// TwinCAT 3 PLC project HAWino
// ProgramVersion: 3.1.4026.19
// libraries:
//   Tc2_Math, * (Beckhoff Automation GmbH)
//   Tc2_Standard, * (Beckhoff Automation GmbH)
//   Tc2_System, * (Beckhoff Automation GmbH)
//   Tc2_Utilities, * (Beckhoff Automation GmbH)
//   Tc3_IotBase, * (Beckhoff Automation GmbH)
//   Tc3_JsonXml, * (Beckhoff Automation GmbH)
//   Tc3_Module, * (Beckhoff Automation GmbH)
// project tree:
//   / BahnplanungTask.TcTTO, MotorTask.TcTTO, PlcTask.TcTTO, SOCTask.TcTTO
//   DUTs/Gewerk 2/ E_RobotState.TcDUT, sCmd.TcDUT, sError.TcDUT, sFahrvektor.TcDUT, sGeneralState.TcDUT, sJob.TcDUT, sJobState.TcDUT, sKoordinate.TcDUT, sMqttIn.TcDUT, sMqttOut.TcDUT, sPosition.TcDUT, sStatesForTest.TcDUT, sToken.TcDUT
//   DUTs/Gewerk 3/ Bumperstatus.TcDUT, EKF_Data.TcDUT, GripperCmd_Enum.TcDUT, Position.TcDUT, ReglerState.TcDUT, RobotControl.TcDUT, RobotStatus.TcDUT, WheelVelocity.TcDUT
//   DUTs/PowerManagement/ FleetManagement.TcDUT, ST_PwrMgmt_HAWino.TcDUT, ST_PwrMgmt_HAWino_In.TcDUT, ST_PwrMgmt_HAWino_Out.TcDUT
//   DUTs/Sys/ CoreDriveState.TcDUT, CoreGripperControlState.TcDUT, DUT_SysState.TcDUT, RobotInternalData.TcDUT, RobotPose.TcDUT, U_IpAdr.TcDUT
//   GVLs/ CollisionDetection.TcGVL, GVL_Gripper.TcGVL, GVL_Maps.TcGVL, GVL_RobotConstant.TcGVL, GVL_Datatransfer23.TcGVL, GVL_RobotCoordinates.TcGVL, MQTT_Bahnplanung_Sync.TcGVL, Var_HAWIno.TcGVL
//   POUs/HAWinoCore/001_MotorTask/ FB_Drehzahlregler.TcPOU, Main_MotorTask.TcPOU, FB_Positionsregler.TcPOU
//   POUs/HAWinoCore/01_Motors/ Bumper.TcPOU, Gripper.TcPOU
//   POUs/HAWinoCore/03_Communication/ Camera.TcPOU, CameraConnectionUDP.TcPOU, MQTT.TcPOU
//   POUs/HAWinoCore/02_IR-Sensors/ IrDistanceFromRaw.TcPOU, IrDistanceSensors.TcPOU
//   POUs/HAWinoCore/04_SystemManagment/ FKT_Scale.TcPOU, PowerManager.TcPOU
//   POUs/HAWinoCore/05_Bahnplanung/ FB_AngleMap.TcPOU, FB_CollisionAvoidance.TcPOU, FB_CollisionAvoidanceV2.TcPOU, FB_CollisionAvoidanceV22.TcPOU, FB_CollisionAvoidanceV3.TcPOU, FB_CollisionAvoidanceV3_4.TcPOU, FB_Mapping.TcPOU, FB_MQTT.TcPOU, FB_MQTTNeu.TcPOU, FB_Navigation.TcPOU, FB_RobotStateMachine.TcPOU, FB_StatesTest.TcPOU, FC_ATAN2.TcPOU, Main_Bahnplanung.TcPOU
//   POUs/HAWinoCore/ HAWino.TcPOU
// real-time tasks:
//   TASK PlcTask: cycle T#10ms, priority 20, ADS port 350
//   TASK MotorTask: cycle T#333us, priority 1, ADS port 354
//   TASK peripherieTask: cycle T#20ms, priority 3, ADS port 351
//   TASK SOCTask: cycle T#5ms, priority 51, ADS port 352
// I/O:
//   DEVICE Gerät 1 (EtherCAT), AmsNetId 5.52.98.210.2.1
//     Klemme 1 (EK1200) [EK1200-5000 EtherCAT Netzteil (2A E-Bus)]
//       Motorklemme A2 (EL7342) [EL7342 2K. DC-Motor-Endstufe (50V, 3.5A)] // Channel 1: Motor 1 | Channel 2: Motor 2
//       Motorklemme A3 (EL7342) [EL7342 2K. DC-Motor-Endstufe (50V, 3.5A)] // Channel 1: Motor 3 | Channel 2: Gripper
//       Digitale Eingänge A4 (EL1008) [EL1008 8K. Dig. Eingang 24V, 3ms]
//       Digitale Ausgänge A5 (EL2004) [EL2004 4K. Dig. Ausgang 24V, 0.5A]
//       Analoge Eingänge A6 (EL3068) [EL3068 8K. Ana. Eingang 0-10V]
//       Analoge Eingänge A7 (EL3104) [EL3104 4K. Ana. Eingang +/-10V Diff.]
//       Temperaturklemme A8 (EL3204) [EL3204 4K. Ana. Eingang PT100 (RTD)]
//       Klemme 9 (EL9011) [EL9011 Endklemme]
//   DEVICE Gerät 2 (RT-Ethernet Adapter)
// variable links:
//   HAWino/HAWino Instance <-> Device 1 (EtherCAT)/Term 1 (EK1200)/Analoge Eingänge A6 (EL3068)
//     PlcTask Inputs/IrDistanceSensors.distanceRaw[{1..8}] <-> AI Standard Channel {1..8}/Value  (8 links)
//   HAWino/HAWino Instance <-> Device 1 (EtherCAT)/Term 1 (EK1200)/Analoge Eingänge A7 (EL3104)
//     PlcTask Inputs/IrDistanceSensors.distanceRaw[9] <-> AI Standard Channel 1/Value
//     SOCTask Inputs/PowerManager.batteryVoltageRaw <-> AI Standard Channel 3/Value
//     SOCTask Inputs/PowerManager.supplyCurrentRaw <-> AI Standard Channel 2/Value
//   HAWino/HAWino Instance <-> Device 1 (EtherCAT)/Term 1 (EK1200)/Digitale Ausgänge A5 (EL2004)
//     SOCTask Outputs/PowerManager.shutdownTrigger <-> InitiateShutdown/Output
//   HAWino/HAWino Instance <-> Device 1 (EtherCAT)/Term 1 (EK1200)/Digitale Eingänge A4 (EL1008)
//     BahnplanungTask Inputs/Bumper.BumperStrip <-> Bumper (S1)/Input
//     BahnplanungTask Inputs/MAIN_Bahnplanung.lightBarrierGripper <-> Channel 6/Input
//     MotorTask Inputs/Gripper.slider <-> Channel 5/Input
//     MotorTask Inputs/Main_MotorTask.bumper <-> Bumper (S1)/Input
//     SOCTask Inputs/Main_MotorTask.sliderGripper <-> Channel 5/Input
//     SOCTask Inputs/PowerManager.shutdownButton <-> ShutdownRequested (S11)/Input
//   HAWino/HAWino Instance <-> Device 1 (EtherCAT)/Term 1 (EK1200)/Motorklemme A2 (EL7342)
//     MotorTask Inputs/Main_MotorTask.currentfromMotor1 <-> DCM Synchron info data Channel 1/Info data 2
//     MotorTask Inputs/Main_MotorTask.currentfromMotor2 <-> DCM Synchron info data Channel 2/Info data 2
//     MotorTask Inputs/Main_MotorTask.n1fromMotor <-> DCM Synchron info data Channel 1/Info data 1
//     MotorTask Inputs/Main_MotorTask.n2fromMotor <-> DCM Synchron info data Channel 2/Info data 1
//     MotorTask Outputs/Main_MotorTask.enableToMotor1 <-> DCM Control Channel 1/Control/Enable
//     MotorTask Outputs/Main_MotorTask.enableToMotor2 <-> DCM Control Channel 2/Control/Enable
//     MotorTask Outputs/Main_MotorTask.velocityToMotor1 <-> DCM Velocity Channel 1/Velocity
//     MotorTask Outputs/Main_MotorTask.velocityToMotor2 <-> DCM Velocity Channel 2/Velocity
//   HAWino/HAWino Instance <-> Device 1 (EtherCAT)/Term 1 (EK1200)/Motorklemme A3 (EL7342)
//     MotorTask Inputs/Main_MotorTask.currentfromMotor3 <-> DCM Synchron info data Channel 1/Info data 2
//     MotorTask Inputs/Main_MotorTask.n3fromMotor <-> DCM Synchron info data Channel 1/Info data 1
//     MotorTask Outputs/Main_MotorTask.enableToMotor3 <-> DCM Control Channel 1/Control/Enable
//     MotorTask Outputs/Main_MotorTask.velocityToMotor3 <-> DCM Velocity Channel 1/Velocity
//     PlcTask Inputs/Gripper.Grippercurrent <-> DCM Synchron info data Channel 2/Info data 2
//     PlcTask Outputs/Gripper.driveEnable <-> DCM Control Channel 2/Control/Enable
//     PlcTask Outputs/Gripper.driveVelocity <-> DCM Velocity Channel 2/Velocity
//   HAWino/HAWino Instance <-> Device 1 (EtherCAT)/Term 1 (EK1200)/Temperaturklemme A8 (EL3204)
//     PlcTask Inputs/MQTT.nBatteryTemperature <-> RTD Inputs Channel 1/Batterytemperature
//   HAWino/HAWino Instance <-> HAWino/HAWino Instance
//     PlcTask Inputs/MQTT.batteryVoltage_V <-> SOCTask Outputs/PowerManager.batteryVoltage_V
//     PlcTask Inputs/MQTT.stMqtt_HAWino_IN/bCheckCurrentDetected <-> SOCTask Outputs/PowerManager.stMqtt_HAWino_IN/bCheckCurrentDetected
//     PlcTask Inputs/MQTT.stMqtt_HAWino_IN/bComCheckAnswer <-> SOCTask Outputs/PowerManager.stMqtt_HAWino_IN/bComCheckAnswer
//     PlcTask Inputs/MQTT.stMqtt_HAWino_IN/fActualBatteryCurrent <-> SOCTask Outputs/PowerManager.stMqtt_HAWino_IN/fActualBatteryCurrent
//     PlcTask Inputs/MQTT.stMqtt_HAWino_IN/fActualBatteryVoltage <-> SOCTask Outputs/PowerManager.stMqtt_HAWino_IN/fActualBatteryVoltage
//     PlcTask Inputs/MQTT.stMqtt_HAWino_IN/fBatteryTemperature <-> SOCTask Outputs/PowerManager.stMqtt_HAWino_IN/fBatteryTemperature
//     PlcTask Inputs/MQTT.stMqtt_HAWino_IN/fSoC <-> SOCTask Outputs/PowerManager.stMqtt_HAWino_IN/fSoC
//     PlcTask Inputs/MQTT.stMqtt_HAWino_IN/nEstimatedChargingTime <-> SOCTask Outputs/PowerManager.stMqtt_HAWino_IN/nEstimatedChargingTime
//     PlcTask Inputs/MQTT.stMqtt_HAWino_IN/nEstimatedRunningTime <-> SOCTask Outputs/PowerManager.stMqtt_HAWino_IN/nEstimatedRunningTime
//     PlcTask Inputs/MQTT.stMqtt_HAWino_IN/nRobotNumber <-> SOCTask Outputs/HAWino.Robot_Number
//     PlcTask Inputs/MQTT.supplyCurrent_A <-> SOCTask Outputs/PowerManager.supplyCurrent_A
//     PlcTask Inputs/MQTT.txtReadInit <-> PlcTask Outputs/HAWino.initDone

CONFIGURATION HAWino
    RESOURCE PLC ON TwinCAT3
        TASK BahnplanungTask(INTERVAL := T#20ms, PRIORITY := 3);
        TASK MotorTask(INTERVAL := T#333us, PRIORITY := 1);
        TASK PlcTask(INTERVAL := T#10ms, PRIORITY := 20);
        TASK SOCTask(INTERVAL := T#5ms, PRIORITY := 51);
        PROGRAM Bumper WITH BahnplanungTask : Bumper;
        PROGRAM MAIN_Bahnplanung WITH BahnplanungTask : MAIN_Bahnplanung;
        PROGRAM Main_MotorTask WITH MotorTask : Main_MotorTask;
        PROGRAM Gripper WITH PlcTask : Gripper;
        PROGRAM HAWino WITH PlcTask : HAWino;
        PROGRAM PowerManager WITH SOCTask : PowerManager;
    END_RESOURCE
END_CONFIGURATION

// ---- DUTs/Gewerk 2/E_RobotState.TcDUT
TYPE E_RobotState :
(
    LoadMaps                    := 0,   // Initial state – load maps, then immediately Standby
    Standby                     := 1,   // Wait for job
    CheckConfirmJob             := 2,   // Check / confirm received job
    SelectMapStart              := 3,   // Select map, write destination to DB, start algorithm
    WaitpointReachedSource      := 4,   // Waitpoint (halt point) reached on source side
    WaitPassiveSource           := 5,   // Halt point occupied – passive wait (source side)
    AlgorithmPreviousSource     := 6,   // Start algorithm to previous target (source side)
    SwitchCoordinatesSource     := 7,   // Switch point coordinates (source side)
    DrivePoint1Align            := 8,   // Drive to point 1 + align angle (from array)
    DrivePoint2Align            := 9,   // Drive to point 2 + align angle
    AtChargingStation           := 10,  // At charging station (branch: job = charging)
    WaitForChargingDone         := 11,  // Charging / wait for done command
    DrivePoint1AfterCharge      := 12,  // Drive to point 1 before station (after charging)
    AtStation                   := 13,  // Arrived at station
    CloseGripper                := 14,  // Close gripper (workpiece present)
    DrivePoint1WithWorkpiece    := 15,  // Drive to point 1 back WITH workpiece
    DrivePoint1NoWorkpiece      := 16,  // Drive to point 1 back WITHOUT workpiece → ParkPos
    DrivePoint3Align            := 17,  // Drive to point 3 + align angle
    DrivePoint4                 := 18,  // Drive to point 4
    ScanRFIDSource              := 19,  // Scan RFID (source) + signal to controller 1
    DrivePoint3ToTarget         := 20,  // Drive to point 3 towards target station
    SelectMapTarget             := 21,  // Select map for target station, write DB, start algorithm
    WaitpointReachedTarget      := 22,  // Waitpoint reached on target side
    WaitPassiveTarget           := 23,  // Halt point occupied – passive wait (target side)
    AlgorithmPreviousTarget     := 24,  // Start algorithm to previous target (target side)
    SwitchCoordinatesTarget     := 25,  // Switch point coordinates (target side)
    DrivePoint5AlignRFID        := 26,  // Drive to point 5 (RFID alignment point) + align
    DrivePoint6AtRFID           := 27,  // Drive to point 6 (at RFID sensor) + align
    ScanRFIDTarget              := 28,  // Scan RFID (target) + signal to controller 1
    DrivePoint5                 := 29,  // Drive to point 5 + align angle
    DrivePoint8BeforeDrop       := 30,  // Drive to point 8 (before drop-off)
    DrivePoint9Drop             := 31,  // Drive to point 9 (drop-off position)
    OpenGripper                 := 32,  // Open gripper
    DrivePoint8AfterDrop        := 33,  // Drive to point 8 (before drop-off – return)
    SelectMapParkPosition       := 34   // Select parking map, output job-done signal
);
END_TYPE

// ---- DUTs/Gewerk 2/sCmd.TcDUT
TYPE sCmd :
STRUCT
	boStop : BOOL;
	boReset :BOOL;
	boJobReset: BOOL;
	boRFIDComplete: BOOL;
	boStartJob : BOOL;
	boTokenGrant :BOOL;
	boCancelCharging: BOOL;
END_STRUCT
END_TYPE

// ---- DUTs/Gewerk 2/sError.TcDUT
TYPE sError :
STRUCT
	boErrorRoutePlanning: BOOL;
	boErrorControl: BOOL;
	boErrorNoWorkpiece: BOOL;
	boErrorWorkpieceLost: BOOL;
END_STRUCT
END_TYPE

// ---- DUTs/Gewerk 2/sFahrvektor.TcDUT
TYPE sFahrvektor :
STRUCT
	reWinkel : REAL;           // Fahrtrichtung
	reGeschwindigkeit : REAL;   // Fahrgeschwindigkeit
END_STRUCT
END_TYPE

// ---- DUTs/Gewerk 2/sGeneralState.TcDUT
TYPE sGeneralState :
STRUCT
	boReady: BOOL;
	boCharging: BOOL;
	strPosition: STRING;
END_STRUCT
END_TYPE

// ---- DUTs/Gewerk 2/sJob.TcDUT
TYPE sJob :
STRUCT
	inJob : INT;
	inJobID : INT;
	inDestination1: INT;
	inDestination2 : INT;
END_STRUCT
END_TYPE

// ---- DUTs/Gewerk 2/sJobState.TcDUT
TYPE sJobState :
STRUCT
	boWorkpieceLoaded: BOOL;
	boTransportWorkpiece: BOOL;
	boJobAccepted: BOOL;
	boWaitForRfidOut: BOOL;
	boWaitForRfidIn: BOOL;
	boWorkpiecePlaced: BOOL;
END_STRUCT
END_TYPE

// ---- DUTs/Gewerk 2/sKoordinate.TcDUT
// =============================================================================
// STRUCT: Koordinatenpunkt (X, Y, Winkel)
// =============================================================================
TYPE sKoordinate :
STRUCT
    rePosX   : REAL;  // X-Koordinate in mm
    rePosY   : REAL;  // Y-Koordinate in mm
    reWinkel : REAL;  // Ausrichtungswinkel in Grad
END_STRUCT
END_TYPE

// ---- DUTs/Gewerk 2/sMqttIn.TcDUT
TYPE sMqttIn :
STRUCT
	sJOB: sJOB;
	sCmd: sCmd;
	boCharging1Connected : BOOL;
	boCharging2Connected : BOOL;
	boNewJob : BOOL;
	END_STRUCT
END_TYPE

// ---- DUTs/Gewerk 2/sMqttOut.TcDUT
TYPE sMqttOut :
STRUCT
	sError: sError;
	sJobState: sJobState;
	sGeneralState: sGeneralState;
	sToken: sToken;
END_STRUCT
END_TYPE

// ---- DUTs/Gewerk 2/sPosition.TcDUT
TYPE sPosition :
STRUCT
	reX 	: LREAL;	// X-Position
	reY 	: LREAL;	// Y-Position
	reWinkel: LREAL; 	// AusrichtungS
END_STRUCT
END_TYPE

// ---- DUTs/Gewerk 2/sStatesForTest.TcDUT
{attribute 'qualified_only'}
{attribute 'strict'}
{attribute 'to_string'}
TYPE sStatesForTest :
(
	Target1Vektor := 0,
	CoordinatesInFrontOfTarget1,
	Wait1,
	Target1,
	Wait2,
	AfterTarget1,
	Target2Vector,
	CoordinatesInFrontOfTarget2,
	Wait3,
	Target2,
	Wait4,
	AfterTarget2,
	ParkingVector,
	Finished
);
END_TYPE

// ---- DUTs/Gewerk 2/sToken.TcDUT
TYPE sToken :
STRUCT
	boTokenRequest: BOOL;
	boTokenRelease: BOOL;
END_STRUCT
END_TYPE

// ---- DUTs/Gewerk 3/Bumperstatus.TcDUT
{attribute 'qualified_only'}
{attribute 'strict'}
TYPE Bumperstatus :
(
	init,
	normal,
	triggered
);
END_TYPE

// ---- DUTs/Gewerk 3/EKF_Data.TcDUT
TYPE EKF_Data : 
	STRUCT
		{attribute 'GUID' := '4651D9AA-F39F-4D87-B1FC-94AB11715483'}
		State : sPosition;
		(*  w1,w2,w3  *)
		wheelSpeed : ARRAY [1..3] OF LREAL;
		P_Start : ARRAY [1..9] OF LREAL;
		timestamp : LREAL;
	END_STRUCT
END_TYPE

// ---- DUTs/Gewerk 3/GripperCmd_Enum.TcDUT
{attribute 'qualified_only'}
{attribute 'strict'}
TYPE GripperCmd_Enum :
(
	noGrip 	:= 0,
	take	:= 1,
	put		:= 2
);
END_TYPE

// ---- DUTs/Gewerk 3/Position.TcDUT
TYPE Position :
	STRUCT
		x, y, theta, e : LREAL; //e = Fehler des Kamerasystems
	END_STRUCT
END_TYPE

// ---- DUTs/Gewerk 3/ReglerState.TcDUT
{attribute 'qualified_only'}
{attribute 'strict'}
TYPE ReglerState :
(
	init,
	idle,
	working,
	stop
);
END_TYPE

// ---- DUTs/Gewerk 3/RobotControl.TcDUT
{attribute 'qualified_only'}
{attribute 'strict'}
{attribute 'to_string'}
TYPE RobotControl :
(
	idle 	:= 0,
	stop 	:= 1,
	reset	:= 2,
	vector	:= 3,
	position := 4
);
END_TYPE

// ---- DUTs/Gewerk 3/RobotStatus.TcDUT
{attribute 'qualified_only'}
{attribute 'strict'}
{attribute 'to_string'}
TYPE RobotStatus :
(
	offline 		:= 0,
	betriebsbereit 	:= 1,
	laufend			:= 2,
	zielErreicht	:= 3,
	fehler			:= 4
);
END_TYPE

// ---- DUTs/Gewerk 3/WheelVelocity.TcDUT
TYPE WheelVelocity :
STRUCT
	wheel1, wheel2, wheel3 : LREAL;
END_STRUCT
END_TYPE

// ---- DUTs/PowerManagement/FleetManagement.TcDUT
TYPE FleetManagement :
STRUCT
	
	nRobotNumber			: INT;
	fSoC					: LREAL;
	nEstimatedRunningTime	: UDINT;
	ChargeRequired			: BOOL;
	
END_STRUCT
END_TYPE

// ---- DUTs/PowerManagement/ST_PwrMgmt_HAWino.TcDUT
TYPE ST_PwrMgmt_HAWino :
STRUCT
	Output	: ST_PwrMgmt_HAWino_In;		// Im Vergleich zur Chargingstation_3 sind hier Input und Output vertauscht!
	Input	: ST_PwrMgmt_HAWino_Out;
END_STRUCT
END_TYPE

// ---- DUTs/PowerManagement/ST_PwrMgmt_HAWino_In.TcDUT
TYPE ST_PwrMgmt_HAWino_In :
STRUCT
	nRobotNumber			: INT;
	tTimestamp				: TIME;		// The smallest unit of time is one millisecond. Example: T#82m47s295ms
	fSoC					: LREAL;
	fActualBatteryCurrent	: LREAL;
	fActualBatteryVoltage	: LREAL;
	fBatteryTemperature		: LREAL;
	nEstimatedRunningTime	: REAL;	
	nEstimatedChargingTime	: REAL;	
	bCheckCurrentDetected	: BOOL;		// 1. Bezeichnung: bNoChargingCurrent
	bComCheckAnswer			: BOOL;		// HAWino answer for communication check
END_STRUCT
END_TYPE

// ---- DUTs/PowerManagement/ST_PwrMgmt_HAWino_Out.TcDUT
TYPE ST_PwrMgmt_HAWino_Out :
STRUCT
	bChargingActive					: BOOL;
	bExternalRecalibrationTrigger	: BOOL;
	fExternalRecalibrationValue		: LREAL;
	bComCheckRequest 				: BOOL;		// Request from charger to HAWino to test stable communication 
END_STRUCT 
END_TYPE

// ---- DUTs/Sys/CoreDriveState.TcDUT
{attribute 'qualified_only'}
{attribute 'strict'}
TYPE CoreDriveState :
(
	Init,
	Drive,
	operational,
	stop,
	error,
	BumperStop
);
END_TYPE

// ---- DUTs/Sys/CoreGripperControlState.TcDUT
{attribute 'qualified_only'}
{attribute 'strict'}
TYPE CoreGripperControlState :
(
	Init,
	Open,
	Closing,
	Closed,
	Opening
);
END_TYPE

// ---- DUTs/Sys/DUT_SysState.TcDUT
{attribute 'qualified_only'}
{attribute 'strict'}
TYPE DUT_SysState :
(
	init:=0,
	preOp:=1,
	Op := 2,
	Error:=3
);
END_TYPE

// ---- DUTs/Sys/RobotInternalData.TcDUT
TYPE RobotInternalData :
	STRUCT
		Robot_Number : INT;
		Robot_IP_WiFi     : T_AmsNetId;
		Robot_IP_Wire     : T_AmsNetId;
		Robot_Name     : STRING;
		Robot_Nickname : STRING;
		factor_V_m : REAL;		// Korrekturfaktor für Spannungsteiler
		sum_V_b	: REAL;			// Korrektursummand für statischen Fehler der Spannung
		factor_I_m : REAL;		// Korrekturfaktor für Strommessung
		sum_I_b	: REAL;			// Korrektursummand für statischen Fehler des Stromes
		
		
	END_STRUCT
END_TYPE

// ---- DUTs/Sys/RobotPose.TcDUT
TYPE RobotPose :
STRUCT
	x, y, theta,e : LREAL;
END_STRUCT
END_TYPE

// ---- DUTs/Sys/U_IpAdr.TcDUT
TYPE U_IpAdr :
UNION
	ipAdrInternal : UDINT;
	ipAdr : ARRAY[0..3] OF BYTE;
END_UNION
END_TYPE

// ---- GVLs/CollisionDetection.TcGVL
{attribute 'qualified_only'}
VAR_GLOBAL CONSTANT
	ANGLE_STATIONARY : LREAL := 999;
	
	NOT_ON_RAIL : INT := 0;
	RAIL_LEFT : INT := 1;
	RAIL_RIGHT : INT := 2;
	
END_VAR

// ---- GVLs/GVL_Gripper.TcGVL
{attribute 'qualified_only'}
VAR_GLOBAL
	cmdGripper : GripperCmd_Enum := GripperCmd_Enum.take;
END_VAR

// ---- GVLs/GVL_Maps.TcGVL
{attribute 'qualified_only'}
VAR_GLOBAL
    sreGoalX : ARRAY[1..13] OF REAL := [49.0, 119.0,  175.0, 250.0,
                                         300.0, 375.0, 430.0, 505.0,
                                         640.0, 100.0, 170.0, 240.0,
                                         310.0];
// 	//Testcase
// 	sreGoalX : ARRAY[1..13] OF REAL := [100.0, 600.0,  186.0, 260.0,
//                                          300.0, 375.0, 430.0, 505.0,
//                                          640.0, 100.0, 150.0, 200.0,
//                                          250.0];									 
// 
//     sreGoalY : ARRAY[1..13] OF REAL := [150.0, 150.0, 288.0, 288.0,
//                                          288.0,  288.0, 288.0, 288.0, 325.0,
//                                          100.0,  100.0, 100.0, 100.0];
										 
 	 sreGoalY : ARRAY[1..13] OF REAL := [288.0, 288.0, 288.0, 288.0,
                                          288.0,  288.0, 288.0, 288.0, 300.0,
                                          100.0,  100.0, 100.0, 100.0];

    stiMapPath : STRING(255) := '/tmp/angle_maps/';
END_VAR

// ---- GVLs/GVL_RobotConstant.TcGVL
{attribute 'qualified_only'}
VAR_GLOBAL CONSTANT
	 ROBOT_RADIUS : LREAL := 0.15;		  // in m
	 RING_SIZE : INT := 60;
END_VAR

// ---- GVLs/GVL_Datatransfer23.TcGVL
{attribute 'qualified_only'}
VAR_GLOBAL
	// Von Gewerk 2 zu Gewerk 3
	gvFahrvektor 	: sFahrvektor;
	gvZielPosition  : sPosition;
	inControl : RobotControl;     // Steuerungsvariable      // 0=idle, 1=Stop, 2=Reset, 3=Vektor, 4=Position
	
	// Von Gewerk 3 zu Gewerk 2
	gvActualPosition	: sPosition;
	inStatus			: RobotStatus; // Statusvariable	// 0=offline, 1=Betriebsbereit, 2=Laufend, 3=Ziel Erreicht, 4=Fehler
END_VAR

// ---- GVLs/GVL_RobotCoordinates.TcGVL
// =============================================================================
// File:        GVL_RobotCoordinates.st
// Description: Global coordinate arrays and index constants for all 4 robots.
//              Pass the matching array to FB_RobotStateMachine.xarstCoordinates.
//              Use the IDX_* constants for all index inputs of the FB.
//
// Usage example in your main program:
//
//   fbHAWino1(
//       xstMqttIn              := stMqttInRobot1,
//       xeRobotStatus          := eStatusRobot1,
//       xboMapsLoaded          := boMapsLoadedRobot1,
//       xboVectorTargetReached := boVectorDoneRobot1,
//       xarstCoordinates       := arstHAWino1,
//       xinSourceIndex         := IDX_STORAGE_1,
//       xinTargetIndex         := IDX_PROD_11,
//       xinRfidSourceIndex     := IDX_RFID_1,
//       xinRfidTargetIndex     := IDX_RFID_3,
//       xinParkingIndex        := IDX_PARKING_101,
//       xinChargingIndex       := IDX_CHARGING_202,
//       xinMapSource           := 1,
//       xinMapTarget           := 3,
//       xinMapParking          := 7
//   );
//
// Array index mapping [0..29]:
//   [0]  Station   1 – Storage 1        [15] Station  42 – Production 42
//   [1]  Station   2 – Storage 2        [16] Station 101 – Parking 1
//   [2]  Station   3 – Storage 3        [17] Station 102 – Parking 2
//   [3]  Station   4 – Storage 4        [18] Station 103 – Parking 3
//   [4]  Station   5 – Drop-off 5       [19] Station 104 – Parking 4
//   [5]  Station   6 – Drop-off 6       [20] Station 201 – Charging 1
//   [6]  Station   7 – Drop-off 7       [21] Station 202 – Charging 2
//   [7]  Station   8 – Drop-off 8       [22] RFID 1
//   [8]  Station  11 – Production 11    [23] RFID 2
//   [9]  Station  12 – Production 12    [24] RFID 3
//   [10] Station  21 – Production 21    [25] RFID 4
//   [11] Station  22 – Production 22    [26] RFID 5
//   [12] Station  31 – Production 31    [27] RFID 6
//   [13] Station  32 – Production 32    [28] RFID 7
//   [14] Station  41 – Production 41    [29] RFID 8
// =============================================================================

VAR_GLOBAL CONSTANT

    IDX_STORAGE_1    : INT := 0;
    IDX_STORAGE_2    : INT := 1;
    IDX_STORAGE_3    : INT := 2;
    IDX_STORAGE_4    : INT := 3;

    IDX_DROPOFF_5    : INT := 4;
    IDX_DROPOFF_6    : INT := 5;
    IDX_DROPOFF_7    : INT := 6;
    IDX_DROPOFF_8    : INT := 7;

    IDX_PROD_11      : INT := 8;
    IDX_PROD_12      : INT := 9;
    IDX_PROD_21      : INT := 10;
    IDX_PROD_22      : INT := 11;
    IDX_PROD_31      : INT := 12;
    IDX_PROD_32      : INT := 13;
    IDX_PROD_41      : INT := 14;
    IDX_PROD_42      : INT := 15;

    IDX_PARKING_101  : INT := 10;
    IDX_PARKING_102  : INT := 11;
    IDX_PARKING_103  : INT := 12;
    IDX_PARKING_104  : INT := 13;

    IDX_CHARGING_201 : INT := 20;
    IDX_CHARGING_202 : INT := 21;

    IDX_RFID_1       : INT := 22;
    IDX_RFID_2       : INT := 23;
    IDX_RFID_3       : INT := 24;
    IDX_RFID_4       : INT := 25;
    IDX_RFID_5       : INT := 26;
    IDX_RFID_6       : INT := 27;
    IDX_RFID_7       : INT := 28;
    IDX_RFID_8       : INT := 29;

END_VAR


VAR_GLOBAL

    // =========================================================================
    // HAWino 1 – xarstCoordinates [0..29]
    // Stations 41/42, Drop-off 5..8, Charging, Parking, RFID: no data yet
    // =========================================================================
    arstHAWino1 : ARRAY[0..29] OF sKoordinate := [
        (rePosX :=  629.6,  rePosY := 2774.6, reWinkel :=    0.5),  // [0]  Storage 1
        (rePosX :=  627.8,  rePosY := 2670.7, reWinkel :=    1.0),  // [1]  Storage 2
        (rePosX := 1061.6,  rePosY := 2779.4, reWinkel :=  179.3),  // [2]  Storage 3
        (rePosX := 1061.3,  rePosY := 2673.0, reWinkel := -179.1),  // [3]  Storage 4
        (rePosX := 4430.4,  rePosY := 2777.9, reWinkel :=    1.2),  // [4]  Drop-off 5  (no data)
        (rePosX := 4430.6,  rePosY := 2668.4, reWinkel :=   -0.8),  // [5]  Drop-off 6  (no data)
        (rePosX := 4855.9,  rePosY := 2774.8, reWinkel := -180.0),  // [6]  Drop-off 7  (no data)
        (rePosX := 4854.4,  rePosY := 2671.2, reWinkel :=  179.3),  // [7]  Drop-off 8  (no data)
        (rePosX := 1904.0,  rePosY := 2768.7, reWinkel :=    0.2),  // [8]  Production 11
        (rePosX := 1902.2,  rePosY := 2669.0, reWinkel :=    1.5),  // [9]  Production 12
        (rePosX := 2341.0,  rePosY := 2767.0, reWinkel := -179.2),  // [10] Production 21
        (rePosX := 2341.3,  rePosY := 2665.1, reWinkel := -179.7),  // [11] Production 22
        (rePosX := 3184.5,  rePosY := 2759.0, reWinkel :=   -0.8),  // [12] Production 31
        (rePosX := 3181.3,  rePosY := 2654.7, reWinkel :=    0.3),  // [13] Production 32
        (rePosX := 3621.4,  rePosY := 2766.4, reWinkel :=  180.0),  // [14] Production 41 (no data)
        (rePosX := 3621.6,  rePosY := 2660.0, reWinkel :=  179.5),  // [15] Production 42 (no data)
        (rePosX :=    0.0,  rePosY :=    0.0, reWinkel :=    0.0),  // [16] Parking 101   (no data)
        (rePosX :=    0.0,  rePosY :=    0.0, reWinkel :=    0.0),  // [17] Parking 102   (no data)
        (rePosX :=    0.0,  rePosY :=    0.0, reWinkel :=    0.0),  // [18] Parking 103   (no data)
        (rePosX :=    0.0,  rePosY :=    0.0, reWinkel :=    0.0),  // [19] Parking 104   (no data)
        (rePosX := 6099.5,  rePosY := 3469.4, reWinkel :=  -21.4),  // [20] Charging 201  (no data)
        (rePosX := 6700.5,  rePosY := 3464.2, reWinkel :=  -19.1),  // [21] Charging 202  (no data)
        (rePosX :=  630.0,  rePosY := 2878.6, reWinkel :=    0.7),  // [22] RFID 1        (no data)
        (rePosX := 1062.2,  rePosY := 2874.4, reWinkel := -178.8),  // [23] RFID 2        (no data)
        (rePosX := 1902.2,  rePosY := 2872.2, reWinkel :=   -0.3),  // [24] RFID 3        (no data)
        (rePosX := 2339.6,  rePosY := 2869.9, reWinkel := -178.5),  // [25] RFID 4        (no data)
        (rePosX := 3186.0,  rePosY := 2866.7, reWinkel :=    0.4),  // [26] RFID 5        (no data)
        (rePosX := 3622.4,  rePosY := 2873.8, reWinkel :=  179.1),  // [27] RFID 6        (no data)
        (rePosX := 4431.6,  rePosY := 2879.1, reWinkel :=    0.6),  // [28] RFID 7        (no data)
        (rePosX := 4857.3,  rePosY := 2876.9, reWinkel := -178.8)   // [29] RFID 8        (no data)
    ];

    // =========================================================================
    // HAWino 2 – xarstCoordinates [0..29]
    // All stations, charging and RFID complete. Parking still no data.
    // =========================================================================
    arstHAWino2 : ARRAY[0..29] OF sKoordinate := [
        (rePosX :=  623.3,  rePosY := 2775.5, reWinkel :=   -0.9),  // [0]  Storage 1
        (rePosX :=  626.9,  rePosY := 2779.0, reWinkel :=    0.2),  // [1]  Storage 2
        (rePosX := 1067.0,  rePosY := 2778.0, reWinkel :=  177.6),  // [2]  Storage 3
        (rePosX := 1065.3,  rePosY := 2668.5, reWinkel := -179.6),  // [3]  Storage 4
        (rePosX := 4425.8,  rePosY := 2777.0, reWinkel :=   -1.1),  // [4]  Drop-off 5
        (rePosX := 4424.3,  rePosY := 2672.8, reWinkel :=    0.0),  // [5]  Drop-off 6
        (rePosX := 4861.3,  rePosY := 2771.6, reWinkel := -180.0),  // [6]  Drop-off 7
        (rePosX := 4860.3,  rePosY := 2673.3, reWinkel :=  178.0),  // [7]  Drop-off 8
        (rePosX := 1894.3,  rePosY := 2771.7, reWinkel :=   -0.3),  // [8]  Production 11
        (rePosX := 1895.3,  rePosY := 2667.8, reWinkel :=    0.0),  // [9]  Production 12
        (rePosX := 2348.3,  rePosY := 2768.7, reWinkel := -179.2),  // [10] Production 21
        (rePosX := 2346.0,  rePosY := 2662.4, reWinkel :=  179.6),  // [11] Production 22
        (rePosX := 3177.3,  rePosY := 2761.7, reWinkel :=    0.8),  // [12] Production 31
        (rePosX := 3173.0,  rePosY := 2647.3, reWinkel :=   -2.9),  // [13] Production 32
        (rePosX := 3629.4,  rePosY := 2763.2, reWinkel := -179.8),  // [14] Production 41
        (rePosX := 3627.7,  rePosY := 2655.2, reWinkel :=  179.7),  // [15] Production 42
        (rePosX :=    0.0,  rePosY :=    0.0, reWinkel :=    0.0),  // [16] Parking 101   (no data)
        (rePosX :=    0.0,  rePosY :=    0.0, reWinkel :=    0.0),  // [17] Parking 102   (no data)
        (rePosX :=    0.0,  rePosY :=    0.0, reWinkel :=    0.0),  // [18] Parking 103   (no data)
        (rePosX :=    0.0,  rePosY :=    0.0, reWinkel :=    0.0),  // [19] Parking 104   (no data)
        (rePosX := 6085.1,  rePosY := 3470.8, reWinkel :=  -19.0),  // [20] Charging 201
        (rePosX := 6726.6,  rePosY := 3468.8, reWinkel :=  -26.7),  // [21] Charging 202
        (rePosX :=  625.5,  rePosY := 2880.0, reWinkel :=   -1.0),  // [22] RFID 1
        (rePosX := 1066.0,  rePosY := 2876.1, reWinkel :=  179.8),  // [23] RFID 2
        (rePosX := 1897.8,  rePosY := 2874.0, reWinkel :=   -0.7),  // [24] RFID 3
        (rePosX := 2345.5,  rePosY := 2870.1, reWinkel := -179.2),  // [25] RFID 4
        (rePosX := 3181.3,  rePosY := 2865.0, reWinkel :=   -1.6),  // [26] RFID 5
        (rePosX := 3629.8,  rePosY := 2868.0, reWinkel := -179.8),  // [27] RFID 6
        (rePosX := 4426.7,  rePosY := 2884.2, reWinkel :=    0.3),  // [28] RFID 7
        (rePosX := 4862.0,  rePosY := 2879.4, reWinkel :=  179.0)   // [29] RFID 8
    ];

    // =========================================================================
    // HAWino 3 – xarstCoordinates [0..29]
    // All stations, charging and RFID complete. Parking still no data.
    // =========================================================================
    arstHAWino3 : ARRAY[0..29] OF sKoordinate := [
        (rePosX :=  629.0,  rePosY := 2774.0, reWinkel :=    0.0),  // [0]  Storage 1
        (rePosX :=  628.1,  rePosY := 2668.6, reWinkel :=    0.4),  // [1]  Storage 2
        (rePosX := 1064.8,  rePosY := 2776.3, reWinkel := -179.7),  // [2]  Storage 3
        (rePosX := 1067.3,  rePosY := 2672.3, reWinkel := -179.6),  // [3]  Storage 4
        (rePosX := 4429.5,  rePosY := 2776.3, reWinkel :=    0.1),  // [4]  Drop-off 5
        (rePosX := 4428.8,  rePosY := 2669.4, reWinkel :=    0.4),  // [5]  Drop-off 6
        (rePosX := 4857.0,  rePosY := 2777.1, reWinkel := -179.7),  // [6]  Drop-off 7
        (rePosX := 4854.4,  rePosY := 2670.3, reWinkel := -179.3),  // [7]  Drop-off 8
        (rePosX := 1902.6,  rePosY := 2766.3, reWinkel :=    0.0),  // [8]  Production 11
        (rePosX := 1902.6,  rePosY := 2668.1, reWinkel :=    1.0),  // [9]  Production 12
        (rePosX := 2341.0,  rePosY := 2772.0, reWinkel :=  179.8),  // [10] Production 21
        (rePosX := 2342.5,  rePosY := 2663.4, reWinkel := -179.2),  // [11] Production 22
        (rePosX := 3183.0,  rePosY := 2760.3, reWinkel :=    0.5),  // [12] Production 31
        (rePosX := 3179.7,  rePosY := 2658.5, reWinkel :=    1.2),  // [13] Production 32
        (rePosX := 3623.4,  rePosY := 2776.0, reWinkel :=  177.6),  // [14] Production 41
        (rePosX := 3622.5,  rePosY := 2663.1, reWinkel :=  178.3),  // [15] Production 42
        (rePosX :=    0.0,  rePosY :=    0.0, reWinkel :=    0.0),  // [16] Parking 101   (no data)
        (rePosX :=    0.0,  rePosY :=    0.0, reWinkel :=    0.0),  // [17] Parking 102   (no data)
        (rePosX :=    0.0,  rePosY :=    0.0, reWinkel :=    0.0),  // [18] Parking 103   (no data)
        (rePosX :=    0.0,  rePosY :=    0.0, reWinkel :=    0.0),  // [19] Parking 104   (no data)
        (rePosX := 6082.9,  rePosY := 3472.0, reWinkel :=  -16.0),  // [20] Charging 201
        (rePosX := 6694.4,  rePosY := 3468.5, reWinkel :=  -16.3),  // [21] Charging 202
        (rePosX :=  629.1,  rePosY := 2877.2, reWinkel :=   -0.1),  // [22] RFID 1
        (rePosX := 1062.3,  rePosY := 2877.4, reWinkel := -179.7),  // [23] RFID 2
        (rePosX := 1902.2,  rePosY := 2872.9, reWinkel :=    0.7),  // [24] RFID 3
        (rePosX := 2340.0,  rePosY := 2872.1, reWinkel := -179.3),  // [25] RFID 4
        (rePosX := 3185.4,  rePosY := 2865.5, reWinkel :=   -0.1),  // [26] RFID 5
        (rePosX := 3624.3,  rePosY := 2872.2, reWinkel :=  179.7),  // [27] RFID 6
        (rePosX := 4430.8,  rePosY := 2877.7, reWinkel :=    0.5),  // [28] RFID 7
        (rePosX := 4858.2,  rePosY := 2882.0, reWinkel :=  179.5)   // [29] RFID 8
    ];

    // =========================================================================
    // HAWino 4 – xarstCoordinates [0..29]
    // All stations, charging and RFID complete. Parking still no data.
    // =========================================================================
    arstHAWino4 : ARRAY[0..29] OF sKoordinate := [
        (rePosX :=  629.7,  rePosY := 2774.1, reWinkel :=   -0.2),  // [0]  Storage 1
        (rePosX :=  628.7,  rePosY := 2669.9, reWinkel :=    0.4),  // [1]  Storage 2
        (rePosX := 1062.0,  rePosY := 2776.0, reWinkel := -179.6),  // [2]  Storage 3
        (rePosX := 1059.0,  rePosY := 2673.0, reWinkel := -179.3),  // [3]  Storage 4
        (rePosX := 4429.6,  rePosY := 2778.1, reWinkel :=    0.0),  // [4]  Drop-off 5
        (rePosX := 4429.0,  rePosY := 2663.4, reWinkel :=   -1.4),  // [5]  Drop-off 6
        (rePosX := 4856.5,  rePosY := 2774.8, reWinkel := -179.8),  // [6]  Drop-off 7
        (rePosX := 4855.7,  rePosY := 2668.8, reWinkel := -179.6),  // [7]  Drop-off 8
        (rePosX := 1903.3,  rePosY := 2770.2, reWinkel :=    0.2),  // [8]  Production 11
        (rePosX := 1902.7,  rePosY := 2666.4, reWinkel :=  -19.8),  // [9]  Production 12
        (rePosX := 2337.0,  rePosY := 2769.3, reWinkel := -179.5),  // [10] Production 21
        (rePosX := 2338.5,  rePosY := 2662.5, reWinkel := -179.0),  // [11] Production 22
        (rePosX := 3183.0,  rePosY := 2762.0, reWinkel :=   -0.3),  // [12] Production 31
        (rePosX := 3182.1,  rePosY := 2656.2, reWinkel :=    0.6),  // [13] Production 32
        (rePosX := 3626.5,  rePosY := 2770.5, reWinkel :=  179.1),  // [14] Production 41
        (rePosX := 3626.6,  rePosY := 2664.2, reWinkel :=  178.6),  // [15] Production 42
        (rePosX :=    0.0,  rePosY :=    0.0, reWinkel :=    0.0),  // [16] Parking 101   (no data)
        (rePosX :=    0.0,  rePosY :=    0.0, reWinkel :=    0.0),  // [17] Parking 102   (no data)
        (rePosX :=    0.0,  rePosY :=    0.0, reWinkel :=    0.0),  // [18] Parking 103   (no data)
        (rePosX :=    0.0,  rePosY :=    0.0, reWinkel :=    0.0),  // [19] Parking 104   (no data)
        (rePosX := 6085.7,  rePosY := 3470.2, reWinkel :=  -17.0),  // [20] Charging 201
        (rePosX := 6701.6,  rePosY := 3468.0, reWinkel :=  -18.4),  // [21] Charging 202
        (rePosX :=  629.2,  rePosY := 2877.5, reWinkel :=    0.0),  // [22] RFID 1
        (rePosX := 1059.6,  rePosY := 2879.0, reWinkel := -179.9),  // [23] RFID 2
        (rePosX := 1900.9,  rePosY := 2877.3, reWinkel :=    1.2),  // [24] RFID 3
        (rePosX := 2337.2,  rePosY := 2871.4, reWinkel := -179.0),  // [25] RFID 4
        (rePosX := 3184.5,  rePosY := 2867.7, reWinkel :=   -0.1),  // [26] RFID 5
        (rePosX := 3623.9,  rePosY := 2870.1, reWinkel :=  179.9),  // [27] RFID 6
        (rePosX := 4430.0,  rePosY := 2876.8, reWinkel :=   -0.5),  // [28] RFID 7
        (rePosX := 4857.7,  rePosY := 2880.0, reWinkel :=  180.0)   // [29] RFID 8
    ];

END_VAR

// ---- GVLs/MQTT_Bahnplanung_Sync.TcGVL
{attribute 'qualified_only'}
VAR_GLOBAL
	
	newJob : BOOL := FALSE;
	critSectionNewJob : FB_IecCriticalSection;
	
	sendCode : BOOL := FALSE;
	critSectionSendCode : FB_IecCriticalSection;
	
	sendMessage : BOOL := FALSE;
	critSectionSendMessage : FB_IecCriticalSection;
	
	sendBumperResetAck : BOOL := FALSE;
	critSectionSendBumperResetAck : FB_IecCriticalSection;
	
	sendPartLostResetAck : BOOL := FALSE;
	critSectionSendPartLostResetAck : FB_IecCriticalSection;
	
	sendGlobalResetAck : BOOL := FALSE;
	critSectionSendGlobalResetAck : FB_IecCriticalSection;
	
END_VAR

// ---- GVLs/Var_HAWIno.TcGVL
// Roboternummern:
// 
// CX-31C9D6 = 1
// CX-35CFB8 = 2
// CX-35CDC8 = 3 
// CX-35CDD6 = 4
// CX-4D0046 = 5

VAR_GLOBAL
	Robot_Number : INT;
END_VAR

// ---- POUs/HAWinoCore/01_Motors/Bumper.TcPOU
PROGRAM Bumper
VAR
	BumperStrip	AT%I*:	BOOL;
	Reset AT%I* : BOOL;
	state: Bumperstatus := Bumperstatus.init;
	Triggered AT%Q* : BOOL;
	R_Reset: R_TRIG;
	
END_VAR


CASE state OF 
	Bumperstatus.init:
		IF NOT BumperStrip AND NOT Reset THEN
			state := Bumperstatus.normal;
		END_IF	
	Bumperstatus.normal:
		IF BumperStrip THEN
			state := Bumperstatus.triggered;
			Triggered := TRUE;
		END_IF				
	Bumperstatus.triggered:
		IF NOT BumperStrip AND R_Reset.Q THEN
			state := Bumperstatus.normal;
			Triggered := FALSE;
		END_IF
END_CASE

END_PROGRAM

// ---- POUs/HAWinoCore/05_Bahnplanung/Main_Bahnplanung.TcPOU
PROGRAM MAIN_Bahnplanung
VAR
    (* 13 Kartenbausteine — jeder hält sein eigenes Array *)
    arfbMaps       : ARRAY[1..14] OF FB_AngleMap;
    fbNav          : FB_Navigation;
	//fbStates	   : FB_StatesTest;
	fbStates : FB_RobotStateMachine;
	fb_mapping : FB_Mapping;
	fb_MQTT : FB_MQTTNeu;//FB_MQTT;

	
    (* Ladesteuerung *)
    inLoadIdx      : INT := 1;
    boAllLoaded    : BOOL := FALSE;
    boLoadError    : BOOL := FALSE;

    (* Navigation *)
    rePosX         : REAL := 180.0;
    rePosY         : REAL :=  20.0;
    inActiveGoal   : INT  :=   1;

    areRobotX      : ARRAY[0..2] OF REAL;
    areRobotY      : ARRAY[0..2] OF REAL;
    aboRobotActive : ARRAY[0..2] OF BOOL;

    reAngleTarget  : REAL;
    reDistToGoal   : REAL;
	reDistFromGoal : REAL;
	reSpeed 	   : REAL;
    boAtGoal       : BOOL;
    boStop         : BOOL;
    boNavError     : BOOL;
	boIdle			: BOOL;
	RobotIndex: INT;
	actualPosX: LREAL;
	actualPosY: LREAL;
	actualPosTheta: LREAL;
	actualError: LREAL;
	boWarning: BOOL;
	reMinDist: REAL;
	sMqttIn : sMqttIn;
	sMqttOut : sMqttOut;
	eStateMachine : E_RobotState;
	sactualKoordinates : sKoordinate;
	lightBarrierGripper AT %I* : BOOL;
	inMqttTokenTargetId : INT;
	_boAwayFromObstacle : BOOL;
	_boPasssiveWait : BOOL;
	_boMovingAway : BOOL;
	_boCharging : BOOL;
	_inChargingStation : INT;
	    reSpeedFactor   : REAL;
    reCurrentSpeed  : REAL;       (* aktuelle Geschwindigkeit — vom Antrieb lesen *)
    reTargetSpeed   : REAL;
	reGoalSlowdown : REAL;
	
    creMaxSpeed     : REAL := 300.0;   (* cm/s *)
	
	boTesthelp : BOOL := TRUE;
	
	TONGripperOpen : TON;
	TONGripperClose : TON;
	boGripperHelp	: BOOL;
	
END_VAR
	
	VAR_TEMP
    tinI : INT; // Temporary variable
	tinJ : INT := 0;
	tarstHAWId: ARRAY[0..29] OF sKoordinate;
	tinSourceIndex          : INT;                          // Array index of source station  (0..21)
    tinTargetIndex          : INT;                          // Array index of target station  (0..21)
    tinRfidSourceIndex      : INT;                          // Array index of RFID point at source (22..29)
    tinRfidTargetIndex      : INT;                          // Array index of RFID point at target (22..29)
    tinParkingIndex         : INT;                          // Array index of parking position (16..19)
    tinChargingIndex        : INT;                          // Array index of charging station (20..21)
	tinMapSource            : INT;                          // Map ID for source station
    tinMapTarget            : INT;                          // Map ID for target station
    tinMapParking           : INT;                          // Map ID for parking position
	tinTargetDirectionIndex : INT;							//
	tinSourceDirectionIndex : INT;
	tinChargingStatus		: INT;
	
	treTestAngle : REAL;
					
	END_VAR

IF NOT boAllLoaded AND NOT boLoadError THEN

    (* Aktuellen Baustein laden *)
    arfbMaps[inLoadIdx](
        xinGoalID := inLoadIdx,
        xboLoad   := TRUE);

    (* Auf Fehler prüfen *)
    IF arfbMaps[inLoadIdx].yboError THEN
        boLoadError := TRUE;
        RETURN;
    END_IF

    (* Wenn fertig: nächste Karte *)
    IF arfbMaps[inLoadIdx].yboDone THEN
        IF inLoadIdx < 14 THEN
            inLoadIdx := inLoadIdx + 1;
        ELSE
            boAllLoaded := TRUE;
        END_IF
    END_IF

    RETURN;   (* Erst navigieren wenn alle Karten geladen *)
END_IF

RobotIndex := Var_HAWIno.Robot_Number;
IF (RobotIndex < 1) OR (RobotIndex > 4) THEN
	// Falls außerhalb Bereich: Default auf 1 setzen 
	RobotIndex := -1;
ELSE
	actualPosX 		:= Camera.cameraData.robotPosition[RobotIndex].x;
	actualPosY 		:= Camera.cameraData.robotPosition[RobotIndex].y;
	actualPosTheta 	:= Camera.cameraData.robotPosition[RobotIndex].theta;
	actualError		:= Camera.cameraData.robotPosition[RobotIndex].e;
END_IF;

FOR tinI := 1 TO 4 BY 1 DO
	IF NOT (RobotIndex = tinI) THEN
   areRobotX[tinJ] := LREAL_TO_REAL(Camera.cameraData.robotPosition[tinI].x) / 10;
   areRobotY[tinJ] := LREAL_TO_REAL(Camera.cameraData.robotPosition[tinI].y) / 10;
   tinJ := tinJ + 1;
   END_IF
END_FOR

FOR tinJ := 0 TO 2 BY 1 DO
IF areRobotX[tinJ] = 0 AND areRobotY[tinJ] = 0 THEN
	aboRobotActive[tinJ] := FALSE;
	ELSE 
		aboRobotActive[tinJ] := TRUE;
	END_IF
END_FOR

sactualKoordinates.rePosX 	:= GVL_Datatransfer23.gvActualPosition.reX / 10;
sactualKoordinates.rePosY 	:= GVL_Datatransfer23.gvActualPosition.reY / 10;
sactualKoordinates.reWinkel := GVL_Datatransfer23.gvActualPosition.reWinkel;


fb_MQTT(xsDataToSend := sMqttOut,
	xsKoordinate :=  sactualKoordinates,
	xboCharging := _boCharging,
	xinChargingPoint := _inChargingStation,
	ysDataToReceive => sMqttIn,
	xinMqttTokenTargetId := inMqttTokenTargetId,
	yinchargingstatus => tinChargingStatus);

(*fbStates (xboVectorTargetReached := boAtGoal,
 xinSatus := GVL_Datatransfer23.inStatus,
 yinControl => GVL_Datatransfer23.inControl,
 ysTargetPosition => GVL_Datatransfer23.gvZielPosition,
 yinTargetMap => inActiveGoal);
*)	
	
	sMqttOut.sJobState.boWorkpieceLoaded := NOT lightBarrierGripper; //TODO Confirm WITH EBEL
	
fb_mapping(
    xstMqttIn              := sMqttIn,
    xinDefaultParkingIndex := IDX_PARKING_101,
	yinSourceDirectionIndex => tinSourceDirectionIndex,
	yinTargetDirectionIndex => tinTargetDirectionIndex,
    yinSourceIndex => tinSourceIndex,
    yinTargetIndex => tinTargetIndex,
    yinRfidSourceIndex => tinRfidSourceIndex,
    yinRfidTargetIndex => tinRfidTargetIndex,
    yinParkingIndex => tinParkingIndex,
    yinChargingIndex => tinChargingIndex,
    yinMapSource => tinMapSource,
    yinMapTarget => tinMapTarget);
	
	
	
CASE RobotIndex OF 
	1:tarstHAWId := arstHAWino1;
	2:tarstHAWId := arstHAWino2;
	3:tarstHAWId := arstHAWino3;
	4:tarstHAWId := arstHAWino4;
END_CASE
	
fbStates (xstMqttIn := sMqttIn, xeRobotStatus := GVL_Datatransfer23.inStatus, 
xboMapsLoaded := boAllLoaded, 
xboVectorTargetReached := boAtGoal, 
xarstCoordinates := tarstHAWId,
xinSourceIndex := tinSourceIndex,
xinSourceDirectionIndex := tinSourceDirectionIndex,
xinTargetDirectionIndex := tinTargetDirectionIndex,
xinTargetIndex := tinTargetIndex,         
xinRfidSourceIndex := tinRfidSourceIndex,
xinRfidTargetIndex := tinRfidTargetIndex,
xinParkingIndex := tinParkingIndex,
xinChargingIndex := tinChargingIndex,
xinMapSource := tinMapSource,
xinMapTarget := tinMapTarget,
xinMapParking := tinParkingIndex,//tinMapParking,
xreDistToGoal := reDistToGoal,
xreDistFromGoal := reDistFromGoal, 
xboWSSensor := NOT lightBarrierGripper,
xboAwayFromObstacle := _boAwayFromObstacle,
xinStatusOfChargin := tinChargingStatus, 
yeControl => GVL_Datatransfer23.inControl,
ystTargetPosition => GVL_Datatransfer23.gvZielPosition,
yinTargetMap => inActiveGoal,
ystMqttOut => sMqttOut,
yeCurrentState => eStateMachine,
yeMqttTokenTargetId => inMqttTokenTargetId,
yboDriveAway => _boMovingAway,
yboPassiveWait => _boPasssiveWait,
yboCharging => _boCharging,
yinCharginStationID => _inChargingStation);

// //TEST COLLISION
// IF boAtGoal AND boTesthelp THEN
// 	inActiveGoal := 2;
// 	boTesthelp := FALSE;
// ELSIF boAtGoal AND NOT boTesthelp THEN
// 	inActiveGoal := 1;
// 	boTesthelp := TRUE;
// END_IF;
// GVL_Datatransfer23.inControl := RobotControl.vector;
// inActiveGoal := 1;
// IF boAtGoal THEN 
// 	GVL_Datatransfer23.inControl := RobotControl.idle;
// ELSE
// GVL_Datatransfer23.inControl := RobotControl.vector;
// END_IF 
// Timer 1: Gripper AUF (closeGripperCommand = FALSE)
(*TONGripperOpen(IN := NOT boGripperHelp, PT := T#5S);

// Timer 2: Gripper ZU (closeGripperCommand = TRUE)  
TONGripperClose(IN := boGripperHelp, PT := T#5S);

// Nach 5s offen → Gripper schließen
IF TONGripperOpen.Q THEN
    boGripperHelp := TRUE;
    Gripper.closeGripperCommand := TRUE;
END_IF

// Nach 5s zu → Gripper öffnen
IF TONGripperClose.Q THEN
    boGripperHelp := FALSE;
    Gripper.closeGripperCommand := FALSE;
END_IF*)

(* ── Navigation ────────────────────────────────────── *)
fbNav(
    xrePosX        := GVL_Datatransfer23.gvActualPosition.reX / 10,
    xrePosY        := GVL_Datatransfer23.gvActualPosition.reY / 10,
    xinGoalID      := inActiveGoal,//14, test for drive away
    xreRobotX      := areRobotX,
    xreRobotY      := areRobotY,
    xboRobotActive := aboRobotActive,
	xboDriveAway   := _boMovingAway, //TRUE, test for driveaway
	xboPassiveWait := _boPasssiveWait,
    xyarMaps       := arfbMaps,
	xreOwnAngle    := reAngleTarget,   (* aktueller Fahrwinkel *)
    xreOwnSpeed    := reCurrentSpeed,   (* aktuelle Geschwindigkeit *)
    yreAngleTarget => reAngleTarget,
    yreDistToGoal  => reDistToGoal,
	yreDistToOldGoal => reDistFromGoal,
    yboAtGoal      => boAtGoal,
    yboStop        => boStop,
	yboWarning     => boWarning,
	yboIdle 		=> boIdle,
    yreMinDist     => reMinDist,
    yboError       => boNavError,
	yboAwayFromStation => _boAwayFromObstacle,
	yreSpeedFactor => reSpeedFactor);
	
	reAngleTarget := - reAngleTarget;
	IF NOT _boPasssiveWait THEN
	IF reDistToGoal < 30 THEN //TODO FINETUNE
		reGoalSlowdown := reDistToGoal /30;
	ELSE
		reGoalSlowdown := 1.0;
	END_IF
	ELSE
		reGoalSlowdown := 1.0;
	END_IF
	IF boAtGoal THEN 
		reSpeed := 0;
	END_IF
	IF _boMovingAway THEN
		reSpeed := 150;
	END_IF
	IF boIdle THEN
		GVL_Datatransfer23.inControl := RobotControl.idle;
	END_IF
	IF boStop THEN
    reTargetSpeed := 0.0;
	ELSE
    reSpeed := creMaxSpeed * reSpeedFactor * reGoalSlowdown;
	END_IF
	
	GVL_Datatransfer23.gvFahrvektor.reGeschwindigkeit := reSpeed;
	GVL_Datatransfer23.gvFahrvektor.reWinkel :=  reAngleTarget;

END_PROGRAM

// ---- POUs/HAWinoCore/05_Bahnplanung/FB_AngleMap.TcPOU
FUNCTION_BLOCK FB_AngleMap
VAR_INPUT
    xinGoalID  : INT;    (* 1..13 — welche Karte dieser Baustein lädt *)
    xboLoad    : BOOL;   (* steigende Flanke startet Ladevorgang      *)
END_VAR
VAR_OUTPUT
    yboDone    : BOOL;
    yboError   : BOOL;
    yinProgress: INT;
END_VAR
VAR
    (* Eigenes Array — nur in dieser Instanz, nicht global *)
    _sarMap      : ARRAY[0..399, 0..799] OF INT;

    _inState     : INT := 0;
    _stiPath     : STRING(255);
    _udExpected  : UDINT := 400 * 800 * 2;
    _fbFileOpen  : FB_FileOpen;
    _fbFileRead  : FB_FileRead;
    _fbFileClose : FB_FileClose;
    _rTrigLoad   : R_TRIG;
END_VAR


(* Flanke auf xboLoad erkennen *)
_rTrigLoad(CLK := xboLoad);

IF _rTrigLoad.Q AND NOT yboDone THEN
    _inState := 0;
    yboDone  := FALSE;
    yboError := FALSE;
END_IF

IF yboDone OR yboError THEN RETURN; END_IF

CASE _inState OF

    0:  (* Pfad aufbauen *)
        IF xinGoalID < 10 THEN
            _stiPath := CONCAT(GVL_Maps.stiMapPath,
                          CONCAT('angle_map_0',
                            CONCAT(TO_STRING(xinGoalID), '.bin')));
        ELSE
            _stiPath := CONCAT(GVL_Maps.stiMapPath,
                          CONCAT('angle_map_',
                            CONCAT(TO_STRING(xinGoalID), '.bin')));
        END_IF

        _fbFileOpen(
            sNetId    := '',
            sPathName := _stiPath,
            nMode     := FOPEN_MODEREAD OR FOPEN_MODEBINARY,
            bExecute  := TRUE);

        _inState := 1;

    1:  (* Warten bis Datei offen *)
        _fbFileOpen(bExecute := FALSE);

        IF _fbFileOpen.bBusy THEN RETURN; END_IF

        IF _fbFileOpen.bError THEN
            yboError := TRUE;
            RETURN;
        END_IF

        _fbFileRead(
            sNetId     := '',
            hFile      := _fbFileOpen.hFile,
            pReadBuff  := ADR(_sarMap[0, 0]),
            cbReadLen  := _udExpected,
            bExecute   := TRUE);

        _inState := 2;

    2:  (* Warten bis Lesen fertig *)
        _fbFileRead(bExecute := FALSE);

        IF _fbFileRead.bBusy THEN RETURN; END_IF

        IF _fbFileRead.bError OR _fbFileRead.cbRead <> _udExpected THEN
            yboError := TRUE;
            RETURN;
        END_IF

        _fbFileClose(
            sNetId   := '',
            hFile    := _fbFileOpen.hFile,
            bExecute := TRUE);

        _inState := 3;

    3:  (* Warten bis Datei geschlossen *)
        _fbFileClose(bExecute := FALSE);

        IF _fbFileClose.bBusy THEN RETURN; END_IF

        yinProgress := 100;
        yboDone     := TRUE;
        _inState    := 4;

    4:  (* Fertig — nichts mehr tun *)
        ;

END_CASE

(* Fortschritt während Laden *)
IF _inState > 0 AND _inState < 4 THEN
    yinProgress := _inState * 25;
END_IF

METHOD GETAngle : INT
VAR_INPUT
    xinPosX : INT;
    xinPosY : INT;
END_VAR
GetAngle := _sarMap[
    MAX(0, MIN(xinPosY, 399)),
    MAX(0, MIN(xinPosX, 799))];
END_METHOD

METHOD GetAngleInterp : REAL
VAR_INPUT
    xrePosX : REAL;
    xrePosY : REAL;
END_VAR
VAR
    _inX0, _inX1 : INT;
    _inY0, _inY1 : INT;
    _reFx, _reFy : REAL;

    _reA00, _reA10 : REAL;
    _reA01, _reA11 : REAL;

    _reSin00, _reSin10 : REAL;
    _reSin01, _reSin11 : REAL;
    _reCos00, _reCos10 : REAL;
    _reCos01, _reCos11 : REAL;

    _reSinInterp : REAL;
    _reCosInterp : REAL;
    _crePI       : REAL := 3.14159265358979;

    (* Hilfsvariablen für korrektes Abschneiden *)
    _reFloorX    : REAL;
    _reFloorY    : REAL;
    _inRaw00     : INT;
    _inRaw10     : INT;
    _inRaw01     : INT;
    _inRaw11     : INT;
END_VAR

(* FLOOR: abschneiden statt runden *)
(* REAL_TO_INT rundet — deshalb manuell mit TRUNC *)
_reFloorX := TRUNC(xrePosX);
_reFloorY := TRUNC(xrePosY);

(* Gebrochene Anteile — immer 0.0 bis <1.0 *)
_reFx := xrePosX - _reFloorX;
_reFy := xrePosY - _reFloorY;

(* Pixelkoordinaten der 4 Eckpunkte *)
_inX0 := MAX(0, MIN(REAL_TO_INT(_reFloorX),     798));
_inX1 := MAX(0, MIN(REAL_TO_INT(_reFloorX) + 1, 799));
_inY0 := MAX(0, MIN(REAL_TO_INT(_reFloorY),     398));
_inY1 := MAX(0, MIN(REAL_TO_INT(_reFloorY) + 1, 399));

(* Rohe INT-Werte aus dem Array *)
_inRaw00 := _sarMap[_inY0, _inX0];
_inRaw10 := _sarMap[_inY0, _inX1];
_inRaw01 := _sarMap[_inY1, _inX0];
_inRaw11 := _sarMap[_inY1, _inX1];

(* Sonderwerte: wenn ein Nachbar Hindernis oder Ziel ist
   → nur den gültigen Pixel verwenden                    *)
IF _inRaw00 = -9999 OR _inRaw00 = -8888 THEN
    _inRaw00 := _inRaw11;
END_IF
IF _inRaw10 = -9999 OR _inRaw10 = -8888 THEN
    _inRaw10 := _inRaw00;
END_IF
IF _inRaw01 = -9999 OR _inRaw01 = -8888 THEN
    _inRaw01 := _inRaw00;
END_IF
IF _inRaw11 = -9999 OR _inRaw11 = -8888 THEN
    _inRaw11 := _inRaw00;
END_IF

(* Winkel in Grad (÷10 wegen Skalierung) *)
_reA00 := INT_TO_REAL(_inRaw00) / 10.0;
_reA10 := INT_TO_REAL(_inRaw10) / 10.0;
_reA01 := INT_TO_REAL(_inRaw01) / 10.0;
_reA11 := INT_TO_REAL(_inRaw11) / 10.0;

(* Sin/Cos der 4 Winkel *)
_reSin00 := SIN(_reA00 * _crePI / 180.0);
_reSin10 := SIN(_reA10 * _crePI / 180.0);
_reSin01 := SIN(_reA01 * _crePI / 180.0);
_reSin11 := SIN(_reA11 * _crePI / 180.0);

_reCos00 := COS(_reA00 * _crePI / 180.0);
_reCos10 := COS(_reA10 * _crePI / 180.0);
_reCos01 := COS(_reA01 * _crePI / 180.0);
_reCos11 := COS(_reA11 * _crePI / 180.0);

(* Bilineare Interpolation *)
_reSinInterp := (1.0 - _reFx) * (1.0 - _reFy) * _reSin00
              + _reFx          * (1.0 - _reFy) * _reSin10
              + (1.0 - _reFx)  * _reFy          * _reSin01
              + _reFx          * _reFy           * _reSin11;

_reCosInterp := (1.0 - _reFx) * (1.0 - _reFy) * _reCos00
              + _reFx          * (1.0 - _reFy) * _reCos10
              + (1.0 - _reFx)  * _reFy          * _reCos01
              + _reFx          * _reFy           * _reCos11;

(* Vektor → Winkel in Grad *)
GetAngleInterp := FC_ATAN2(
                    xreY := _reSinInterp,
                    xreX := _reCosInterp)
                  * 180.0 / _crePI;
END_METHOD

END_FUNCTION_BLOCK

// ---- POUs/HAWinoCore/05_Bahnplanung/FC_ATAN2.TcPOU
FUNCTION FC_ATAN2 : REAL
VAR_INPUT
    xreY : REAL;
    xreX : REAL;
END_VAR
VAR
    _crePI : REAL := 3.14159265358979;
END_VAR


IF xreX > 0.0 THEN
    FC_ATAN2 := ATAN(xreY / xreX);

ELSIF xreX < 0.0 AND xreY >= 0.0 THEN
    FC_ATAN2 := ATAN(xreY / xreX) + _crePI;

ELSIF xreX < 0.0 AND xreY < 0.0 THEN
    FC_ATAN2 := ATAN(xreY / xreX) - _crePI;

ELSIF xreX = 0.0 AND xreY > 0.0 THEN
    FC_ATAN2 := _crePI / 2.0;

ELSIF xreX = 0.0 AND xreY < 0.0 THEN
    FC_ATAN2 := -(_crePI / 2.0);

ELSE
    FC_ATAN2 := 0.0;
END_IF

END_FUNCTION

// ---- POUs/HAWinoCore/05_Bahnplanung/FB_Navigation.TcPOU
FUNCTION_BLOCK FB_Navigation
VAR_INPUT
    xrePosX        : REAL;
    xrePosY        : REAL;
    xinGoalID      : INT;
    xreRobotX      : ARRAY[0..2] OF REAL;
    xreRobotY      : ARRAY[0..2] OF REAL;
    xboRobotActive : ARRAY[0..2] OF BOOL;
    (* NEU: Betriebsmodi *)
    xboPassiveWait : BOOL;   (* TRUE = Roboter wartet passiv, weicht fahrenden Robbys aus *)
    xboDriveAway   : BOOL;   (* TRUE = Roboter faehrt aktiv vom Hindernis weg via Ortho-Karte *)
	xreOwnAngle : REAL;
	xreOwnSpeed : REAL;
END_VAR
VAR_OUTPUT
    yreAngleTarget  : REAL;
    yreDistToGoal   : REAL;
    yboAtGoal       : BOOL;
    yboStop         : BOOL;
    yboError        : BOOL;
    yboWarning      : BOOL;
    yreMinDist      : REAL;
    yreDistToOldGoal: REAL;
	yboIdle			: BOOL;
    (* NEU: Ausgaenge *)
    yboAwayFromStation : BOOL;  (* TRUE sobald Ortho-Einflussbereich verlassen (-7777) *)
    yboMovingAway      : BOOL;  (* TRUE wenn im PassiveWait-Modus ein anderer Robby nah ist *)
	yreSpeedFactor : REAL;   (* neu: 0.0..1.0 *)
END_VAR
VAR_IN_OUT
    xyarMaps : ARRAY[1..14] OF FB_AngleMap;
END_VAR
VAR
    _fbCollision    : FB_CollisionAvoidanceV3;
	_fbCollisionPassive    : FB_CollisionAvoidanceV3;
    _inPosX         : INT;
    _inPosY         : INT;
    _reRawAngle     : REAL;
    _reStatGx       : REAL;
    _reStatGy       : REAL;
    _reDynGx        : REAL;
    _reDynGy        : REAL;
    _reTotalGx      : REAL;
    _reTotalGy      : REAL;
    _reDiffX        : REAL;
    _reDiffY        : REAL;
    _reDist         : REAL;
    _reDistSq       : REAL;
    _reLastAngle    : REAL := 0.0;
    _reDelta        : REAL;
    _reAngleRaw     : REAL;
    _inIdx          : INT := 0;
    _inOldGoalID    : INT := 0;
    _inHelperOldGoal: INT := 0;
 
    (* NEU: interne Variablen fuer Ortho-Karte und PassiveWait *)
    _inOrthoRaw     : INT;   (* Rohwert aus Ortho-Karte (x10 Grad) *)
    _reOrthoAngle   : REAL;  (* Umgerechneter Winkel in Grad *)
    _reOrthoGx      : REAL;
    _reOrthoGy      : REAL;
    _rePassiveGx    : REAL;
    _rePassiveGy    : REAL;
    _reNearRobotDist: REAL;  (* kuerzester Abstand zu einem aktiven, fahrenden Robby *)
    _i              : INT;
    _reDx           : REAL;
    _reDy           : REAL;
 
    _crePI              : REAL := 3.14159265358979;
    _creRepulseK        : REAL := 1000.0;
    _creRepulseRad      : REAL := 500.0;
    _creStopDist        : REAL := 5.0;
    _creGoalRadius      : REAL := 5.0;
    _creMaxDeltaDeg     : REAL := 2.0; //2
    (* NEU: Schwellwert – ab welchem Abstand ein naher Robby als "zu nah" gilt (PassiveWait) *)
    _crePassiveTrigDist : REAL := 80.0;   (* Pixel, anpassen nach Bedarf *)
    (* Index der Ortho-Karte im xyarMaps-Array *)
    _cinPassiveMap      : INT := 14;
END_VAR

(* ══════════════════════════════════════════════════════════════
   ZIEL-ID-TRACKING (unveraendert)
   ══════════════════════════════════════════════════════════════ *)
IF xinGoalID <> _inHelperOldGoal THEN
    _inOldGoalID     := _inHelperOldGoal;
    _inHelperOldGoal := xinGoalID;
END_IF
 
(* ── Ausgaenge zuruecksetzen ──────────────────────────────── *)
yboAwayFromStation := FALSE;
yboMovingAway      := FALSE;
yboIdle 		   := FALSE;
(* ══════════════════════════════════════════════════════════════
   MODUS: xboDriveAway
   Roboter faehrt aktiv weg – Ortho-Karte (Map 11) steuert.
   Sobald der Ortho-Einflussbereich verlassen wird (-7777),
   wird yboAwayFromStation = TRUE gesetzt.
   ══════════════════════════════════════════════════════════════ *)
IF xboDriveAway THEN
 
    (* Eingaben pruefen: Ortho-Karte muss geladen sein *)
    IF NOT xyarMaps[_cinPassiveMap].yboDone THEN
        yboError := TRUE; RETURN;
    END_IF
    yboError := FALSE;
 
    (* Koordinaten begrenzen *)
    _inPosX := REAL_TO_INT(TRUNC(xrePosX));
    _inPosY := REAL_TO_INT(TRUNC(xrePosY));
    _inPosX := MAX(0, MIN(_inPosX, 799));
    _inPosY := MAX(0, MIN(_inPosY, 399));
 
    (* Rohwert aus Ortho-Karte lesen *)
    _inOrthoRaw := xyarMaps[_cinPassiveMap].GetAngle(
                       xinPosX := _inPosX,
                       xinPosY := _inPosY);
 
    (* Sonderwert -9999: Hindernis – Notstopp *)
    IF _inOrthoRaw = -9999 THEN
        yboStop := TRUE; RETURN;
    END_IF
 
    (* Sonderwert -7777: ausserhalb Einflussbereich -> Signal setzen, Roboter anhalten *)
    IF _inOrthoRaw = -7777 THEN
        yboAwayFromStation := TRUE;
        yboIdle            := TRUE;   (* Fahrt stoppen, uebergeordnete SPS entscheidet weiter *)
        yreAngleTarget     := _reLastAngle;
        RETURN;
    END_IF
 
    (* Gueltiger Ortho-Winkel: Fahrtrichtung setzen *)
    _reOrthoAngle  := INT_TO_REAL(_inOrthoRaw) / 10.0;   (* /10 wegen Faktor-10-Skalierung *)
 
    (* Kollisionsvermeidung auch im DriveAway-Modus aktiv *)
    _fbCollision(
        xrePosX        := xrePosX,
        xrePosY        := xrePosY,
        xreRobotX      := xreRobotX,
        xreRobotY      := xreRobotY,
        xboRobotActive := xboRobotActive,
		xreOwnAngle    := xreOwnAngle,
		xreOwnSpeed := xreOwnSpeed);
    yboWarning := _fbCollision.yboWarning;
    yreMinDist := _fbCollision.yreMinDist;
	yreSpeedFactor := _fbCollision.yreSpeedFactor;
 
    IF _fbCollision.yboStop THEN
        yboStop        := TRUE;
        yreAngleTarget := THIS^.LimitAngleRate(
                            xreAngleRaw    := _reOrthoAngle,
                            xreMaxDeltaDeg := _creMaxDeltaDeg);
        RETURN;
    END_IF
    yboStop := FALSE;
 
    (* Superposition: Ortho-Vektor + Kollisionsvermeidung *)
    _reOrthoGx := COS(_reOrthoAngle * _crePI / 180.0);
    _reOrthoGy := SIN(_reOrthoAngle * _crePI / 180.0);
    _reTotalGx := _reOrthoGx + _fbCollision.yreDynGx;
    _reTotalGy := _reOrthoGy + _fbCollision.yreDynGy;
 
    IF TRUE THEN //SQRT(_reTotalGx * _reTotalGx + _reTotalGy * _reTotalGy) < 0.001 THEN
        yreAngleTarget := _reOrthoAngle;//THIS^.LimitAngleRate(
                            //xreAngleRaw    := _reOrthoAngle,
                            //xreMaxDeltaDeg := _creMaxDeltaDeg);
    ELSE
        yreAngleTarget := THIS^.LimitAngleRate(
                            xreAngleRaw    := FC_ATAN2(
                                                xreY := _reTotalGy,
                                                xreX := _reTotalGx) * 180.0 / _crePI,
                            xreMaxDeltaDeg := _creMaxDeltaDeg);
    END_IF
 		(*IF (yreAngleTarget < -90) OR (yreAngleTarget > 90) THEN
			yreAngleTarget := 180;
		ELSE
			yreAngleTarget := 0;
		END_IF*)
		(*IF (xinGoalID = 1) OR (xinGoalID = 3) OR (xinGoalID = 5) OR (xinGoalID = 7) THEN
			yreAngleTarget := 180;
		ELSE
			yreAngleTarget := 0;
		END_IF*)
		
    RETURN;   (* DriveAway-Modus abgeschlossen, Rest ueberspringen *)
END_IF
 
(* ══════════════════════════════════════════════════════════════
   MODUS: xboPassiveWait
   Roboter steht still. Naehert sich ein fahrender Robby,
   weicht er mit Hilfe der Ortho-Karte aus (yboMovingAway=TRUE).
   ══════════════════════════════════════════════════════════════ *)
IF xboPassiveWait THEN
 
    IF NOT xyarMaps[_cinPassiveMap].yboDone THEN
        yboError := TRUE; RETURN;
    END_IF
    yboError := FALSE;
 
    (* Abstand zum naechsten AKTIVEN (= fahrenden) Roboter ermitteln *)
    _reNearRobotDist := 1.0E+9;
    FOR _i := 0 TO 2 DO
        IF xboRobotActive[_i] THEN
            _reDx := xrePosX - xreRobotX[_i];
            _reDy := xrePosY - xreRobotY[_i];
            _reDist := SQRT(_reDx * _reDx + _reDy * _reDy);
            IF _reDist < _reNearRobotDist THEN
                _reNearRobotDist := _reDist;
            END_IF
        END_IF
    END_FOR
    yreMinDist := _reNearRobotDist;
 
    (* Kein fahrender Robby in der Naehe -> stehen bleiben *)
    IF _reNearRobotDist > _crePassiveTrigDist THEN
        yboIdle        := TRUE;
        yreAngleTarget := _reLastAngle;   (* Winkel einfrieren *)
        RETURN;
    END_IF
 
    (* Fahrender Robby zu nah -> Ortho-Karte zum Ausweichen nutzen *)
    yboMovingAway := TRUE;
 
    _inPosX := REAL_TO_INT(TRUNC(xrePosX));
    _inPosY := REAL_TO_INT(TRUNC(xrePosY));
    _inPosX := MAX(0, MIN(_inPosX, 799));
    _inPosY := MAX(0, MIN(_inPosY, 399));
 
    _inOrthoRaw := xyarMaps[_cinPassiveMap].GetAngle(
                       xinPosX := _inPosX,
                       xinPosY := _inPosY);
 
    (* Hinderniszelle oder ausserhalb Einflussbereich: Notbremse *)
    IF _inOrthoRaw = -9999 THEN
        yboIdle        := TRUE;
        yreAngleTarget := _reLastAngle;
        RETURN;
    END_IF
 
    _reOrthoAngle := INT_TO_REAL(_inOrthoRaw) / 10.0;
 
    (* Kollisionsvermeidung gegenueber anderen Robbys *)
    _fbCollisionPassive(
        xrePosX        := xrePosX,
        xrePosY        := xrePosY,
        xreRobotX      := xreRobotX,
        xreRobotY      := xreRobotY,
        xboRobotActive := xboRobotActive,
		xreOwnAngle    := xreOwnAngle,
		xreOwnSpeed := xreOwnSpeed);
     yboWarning := _fbCollisionPassive.yboWarning;
    yreMinDist := _fbCollisionPassive.yreMinDist;
	yreSpeedFactor := _fbCollisionPassive.yreSpeedFactor;
 
    IF _fbCollisionPassive.yboStop THEN
        yboStop        := TRUE;
        yreAngleTarget := THIS^.LimitAngleRate(
                            xreAngleRaw    := _reOrthoAngle,
                            xreMaxDeltaDeg := _creMaxDeltaDeg);
        RETURN;
    END_IF
    yboStop := FALSE;
 	IF _inOrthoRaw = -7777 THEN
	_reTotalGx := _fbCollisionPassive.yreDynGx;
    _reTotalGy := _fbCollisionPassive.yreDynGy;
	ELSE
    _reOrthoGx := COS(_reOrthoAngle * _crePI / 180.0);
    _reOrthoGy := SIN(_reOrthoAngle * _crePI / 180.0);
    _reTotalGx := _reOrthoGx + _fbCollisionPassive.yreDynGx;
    _reTotalGy := _reOrthoGy + _fbCollisionPassive.yreDynGy;
 END_IF

        yreAngleTarget := THIS^.LimitAngleRate(
                            xreAngleRaw    := FC_ATAN2(
                                                xreY := _reTotalGy,
                                                xreX := _reTotalGx) * 180.0 / _crePI,
                            xreMaxDeltaDeg := _creMaxDeltaDeg);
 
    RETURN;   (* PassiveWait-Modus abgeschlossen *)
END_IF
 
(* ══════════════════════════════════════════════════════════════
   NORMALBETRIEB: Zielnavigation (unveraendert)
   ══════════════════════════════════════════════════════════════ *)
IF xinGoalID < 1 OR xinGoalID > 13 THEN
    yboError := TRUE; RETURN;
END_IF
IF NOT xyarMaps[xinGoalID].yboDone THEN
    yboError := TRUE; RETURN;
END_IF
yboError := FALSE;

(* ── 1) Abstand zum Ziel ───────────────────────────────────── *)
_reDiffX      := xrePosX - GVL_Maps.sreGoalX[xinGoalID];
_reDiffY      := xrePosY - GVL_Maps.sreGoalY[xinGoalID];
yreDistToGoal := SQRT(_reDiffX * _reDiffX + _reDiffY * _reDiffY);
 
IF _inOldGoalID <> 0 THEN
    _reDiffX         := xrePosX - GVL_Maps.sreGoalX[_inOldGoalID];
    _reDiffY         := xrePosY - GVL_Maps.sreGoalY[_inOldGoalID];
    yreDistToOldGoal := SQRT(_reDiffX * _reDiffX + _reDiffY * _reDiffY);
END_IF
 
(* ── 2) Ziel erreicht? ─────────────────────────────────────── *)
IF yreDistToGoal <= _creGoalRadius THEN
    yboAtGoal      := TRUE;
    yreAngleTarget := 0.0;
    RETURN;
END_IF
yboAtGoal := FALSE;
 
(* ── 3) Koordinaten begrenzen ──────────────────────────────── *)
_inPosX := REAL_TO_INT(TRUNC(xrePosX));
_inPosY := REAL_TO_INT(TRUNC(xrePosY));
_inPosX := MAX(0, MIN(_inPosX, 799));
_inPosY := MAX(0, MIN(_inPosY, 399));
 
(* ── 4) Hindernischeck ─────────────────────────────────────── *)
IF xyarMaps[xinGoalID].GetAngle(
       xinPosX := _inPosX,
       xinPosY := _inPosY) = -9999 THEN
    yboStop := TRUE; RETURN;
END_IF
 
(* ── 5) Winkel aus Karte ────────────────────────────────────── *)
_reRawAngle := xyarMaps[xinGoalID].GetAngleInterp(
                   xrePosX := xrePosX,
                   xrePosY := xrePosY);
_reStatGx := COS(_reRawAngle * _crePI / 180.0);
_reStatGy := SIN(_reRawAngle * _crePI / 180.0);
 
(* ── 6) Kollisionsvermeidung ───────────────────────────────── *)
_fbCollision(
    xrePosX        := xrePosX,
    xrePosY        := xrePosY,
    xreRobotX      := xreRobotX,
    xreRobotY      := xreRobotY,
    xboRobotActive := xboRobotActive,
	xreOwnAngle    := xreOwnAngle,
	xreOwnSpeed := xreOwnSpeed,
	xinOwnID := Robot_Number);
yboWarning := _fbCollision.yboWarning;
yreMinDist := _fbCollision.yreMinDist;
yreSpeedFactor := _fbCollision.yreSpeedFactor;
 
(* ── 7) Notstopp ───────────────────────────────────────────── *)
IF _fbCollision.yboStop THEN
    yboStop        := TRUE;
    yreAngleTarget := THIS^.LimitAngleRate(
                        xreAngleRaw    := _reRawAngle,
                        xreMaxDeltaDeg := _creMaxDeltaDeg);
    RETURN;
END_IF
yboStop := FALSE;
 
(* ── 8) Superposition ──────────────────────────────────────── *)
_reTotalGx := _reStatGx + _fbCollision.yreDynGx;
_reTotalGy := _reStatGy + _fbCollision.yreDynGy;
 
(* ── 9) Winkelberechnung + Rate Limiter ────────────────────── *)
IF SQRT(_reTotalGx * _reTotalGx + _reTotalGy * _reTotalGy) < 0.001 THEN
    yreAngleTarget := THIS^.LimitAngleRate(
                        xreAngleRaw    := _reRawAngle,
                        xreMaxDeltaDeg := _creMaxDeltaDeg);
ELSE
    yreAngleTarget := THIS^.LimitAngleRate(
                        xreAngleRaw    := FC_ATAN2(
                                            xreY := _reTotalGy,
                                            xreX := _reTotalGx)
                                          * 180.0 / _crePI,
                        xreMaxDeltaDeg := _creMaxDeltaDeg);
END_IF

METHOD LimitAngleRate : REAL
VAR_INPUT
    xreAngleRaw     : REAL;   (* neuer ungbegrenzter Winkel *)
    xreMaxDeltaDeg  : REAL;   (* max. Änderung pro Zyklus   *)
END_VAR
VAR
    _reDelta : REAL;
    _reResult: REAL;
END_VAR
IF _reLastAngle = 0 THEN
	_reLastAngle := xreAngleRaw;
END_IF
(* ── Winkeldifferenz berechnen ─────────────────────── *)
_reDelta := xreAngleRaw - _reLastAngle;

(* ── Auf [-180, +180] normieren ────────────────────── *)
WHILE _reDelta > 180.0 DO
    _reDelta := _reDelta - 360.0;
END_WHILE
WHILE _reDelta < -180.0 DO
    _reDelta := _reDelta + 360.0;
END_WHILE

IF (ABS(_reDelta) > 180) THEN
	_reLastAngle := xreAngleRaw;
	LimitAngleRate := xreAngleRaw;
	RETURN;
END_IF


(* ── Änderung begrenzen ─────────────────────────────── *)
IF _reDelta > xreMaxDeltaDeg THEN
    _reDelta := xreMaxDeltaDeg;
ELSIF _reDelta < -xreMaxDeltaDeg THEN
    _reDelta := -xreMaxDeltaDeg;
END_IF

(* ── Neuen Winkel berechnen ─────────────────────────── *)
_reResult := _reLastAngle + _reDelta;

(* ── Auf [-180, +180] halten ────────────────────────── *)
IF _reResult > 180.0 THEN
    _reResult := _reResult - 360.0;
ELSIF _reResult < -180.0 THEN
    _reResult := _reResult + 360.0;
END_IF

(* ── Für nächsten Zyklus speichern ─────────────────── *)
_reLastAngle := _reResult;

LimitAngleRate := _reResult;
END_METHOD

END_FUNCTION_BLOCK

// ---- POUs/HAWinoCore/05_Bahnplanung/FB_CollisionAvoidanceV3.TcPOU
FUNCTION_BLOCK FB_CollisionAvoidanceV3
VAR_INPUT
    xrePosX        : REAL;
    xrePosY        : REAL;
    xreOwnAngle    : REAL;
    xreOwnSpeed    : REAL;
    xreRobotX      : ARRAY[0..2] OF REAL;
    xreRobotY      : ARRAY[0..2] OF REAL;
    xboRobotActive : ARRAY[0..2] OF BOOL;
	xinOwnID : INT;
END_VAR
VAR_OUTPUT
    yreDynGx           : REAL;
    yreDynGy           : REAL;
    yboStop            : BOOL;
    yboWarning         : BOOL;
    yreMinDist         : REAL;
    yreSpeedFactor     : REAL;
    yreNearestRobotDir : REAL;
	yreAusgangsTest : REAL;
END_VAR
VAR
    _inIdx         : INT;
    _reDiffX       : REAL;
    _reDiffY       : REAL;
    _reDist        : REAL;
    _reRepulse     : REAL;
    _reNearestDist : REAL;
	
	_arDist : ARRAY[0..2] OF REAL;

	
	rToleranz        : REAL := 5.0; (* Dein "Bereich", z.B. 5 Grad *)
    rDifferenz       : REAL;
    bImBereich       : BOOL;
	
	
	_reCross      : REAL;
_reFrontal    : REAL;
_rePerpX      : REAL;
_rePerpY      : REAL;
_rePerpWeight : REAL;
_aboPerpActive : ARRAY[0..2] OF BOOL;   (* Latch pro Roboter *)

    (* Lokale Koordinaten für Bias *)
    _reOwnRad      : REAL;
    _reFwdX        : REAL;
    _reFwdY        : REAL;
    _reRightX      : REAL;
    _reRightY      : REAL;
    _reLong        : REAL;
    _reLat         : REAL;

    (* ── Tuning — nur diese 6 Parameter ───────────── *)
    _creRepulseRad  : REAL := 90.0;   (* Wirkradius in cm                  *) //70  alt aber weit entfernt    50 ziemlich dicht aber langsam
    _creRepulseK    : REAL := 3000;//3000 (* Abstoßungskraft                   *)
    _creStopDist    : REAL := 20.0;   (* Notstopp in cm                    *)
    _creWarnDist    : REAL := 45.0;   (* Warnung in cm                     *) //macht glaube nichts ???
    _creSlowDist    : REAL := 60.0;   (* Abbremsen ab hier    100             *)
    _creRightBias   : REAL := 2.0;   (* Rechtsversatz 0=kein Bias, 1=viel *)

END_VAR

(* ── Reset ─────────────────────────────────────────── *)
yreDynGx           := 0.0;
yreDynGy           := 0.0;
yboStop            := FALSE;
yboWarning         := FALSE;
yreMinDist         := 9999.0;
yreSpeedFactor     := 1.0;
yreNearestRobotDir := 0.0;
_reNearestDist     := 9999.0;

(* ── Fahrtrichtung ──────────────────────────────────── *)
_reOwnRad := xreOwnAngle * 3.14159265 / 180.0;
_reFwdX   :=  COS(_reOwnRad);
_reFwdY   :=  SIN(_reOwnRad);
_reRightX :=  SIN(_reOwnRad);
_reRightY := -COS(_reOwnRad);

FOR _inIdx := 0 TO 2 DO
    IF NOT xboRobotActive[_inIdx] THEN CONTINUE; END_IF

    (* ── Abstand ───────────────────────────────────── *)
    _reDiffX := xrePosX - xreRobotX[_inIdx];
    _reDiffY := xrePosY - xreRobotY[_inIdx];
    _reDist  := SQRT(_reDiffX * _reDiffX + _reDiffY * _reDiffY);
	_arDist[_inIdx] := _reDist;
    IF _reDist < 0.1 THEN CONTINUE; END_IF

    (* ── Nächsten Roboter ───────────────────────────── *)
    IF _reDist < _reNearestDist THEN
        _reNearestDist     := _reDist;
        yreMinDist         := _reDist;
        yreNearestRobotDir := FC_ATAN2(
                                xreY := -_reDiffY,
                                xreX := -_reDiffX)
                              * 180.0 / 3.14159265;
    END_IF

    (* ── Zonen ─────────────────────────────────────── *)
    IF _reDist < _creStopDist  THEN yboStop    := TRUE; END_IF
    IF _reDist < _creWarnDist  THEN yboWarning := TRUE; END_IF

    (* ── Geschwindigkeitsreduktion ─────────────────── *)
    IF _reDist < _creSlowDist THEN
        IF _reDist <= _creStopDist THEN
            yreSpeedFactor := 0.0;
        ELSE
            yreSpeedFactor := MIN(
                yreSpeedFactor,
                (_reDist - _creStopDist) /
                ( 1.05 * _creSlowDist - _creStopDist));
        END_IF
    END_IF

    (* ── Außerhalb Wirkradius ───────────────────────── *)
    IF _reDist > _creRepulseRad THEN CONTINUE; END_IF

    (* ── Projektion ─────────────────────────────────── *)
    _reLong := -(_reDiffX * _reFwdX   + _reDiffY * _reFwdY);
    _reLat  := -(_reDiffX * _reRightX + _reDiffY * _reRightY);

    (* ── Nur reagieren wenn Roboter vor uns ist ─────── *)
    (* Hinter uns: halbe Kraft                           *)
    IF _reLong < 0.0 THEN
        _reRepulse := (_creRepulseK / MAX(_reDist * _reDist, 1.0)) * 0.5;
    ELSE
        _reRepulse := _creRepulseK / MAX(_reDist * _reDist, 1.0) ;
    END_IF

    (* ── Geschwindigkeit skaliert Kraft ─────────────── *)
    _reRepulse := MAX(_reRepulse *
                  (1.0 + (xreOwnSpeed / 80.0) * 0.8), 1.1);//1.2

				  
    (* ── Abstoßungsvektor in Weltkoordinaten ────────── *)
    (* Direkte Abstoßung: weg vom anderen Roboter        *)
    yreDynGx := yreDynGx + _reRepulse * _reDiffX / _reDist;
    yreDynGy := yreDynGy + _reRepulse * _reDiffY / _reDist;
	
	

// //     (* ── Rechts-Bias: feste Komponente nach rechts ──── *)
// //     (* Nur wenn Roboter vor uns (_reLong > 0)            *)
// //     (* Stärker wenn Roboter links (_reLat < 0)           *)
// // 
// //  // 1. Differenz berechnen
// // rDifferenz := yreNearestRobotDir - xreOwnAngle;
// // // 2. Normierung auf den Bereich [-180, 180]
// // // Das fängt den Sprung bei +/- 180 Grad ab
// // WHILE rDifferenz > 180.0 DO
// //     rDifferenz := rDifferenz - 360.0;
// // END_WHILE;
// // WHILE rDifferenz <= -180.0 DO
// //     rDifferenz := rDifferenz + 360.0;
// // END_WHILE;
// // // 3. Prüfen, ob man innerhalb der "Breite" liegt
// // IF ABS(rDifferenz) <= rToleranz THEN
// //     bImBereich := TRUE;
// // ELSE
// //     bImBereich := FALSE;
// // END_IF;
// // 
// // 	//IF bImBereich = TRUE THEN
// //    // IF _reLong > 0.0 THEN
// //       //  yreDynGx := yreDynGx + _reRightX * _reRepulse * _creRightBias *_reDiffX / _reDist;
// //                //    * MAX(0.0, 1.0 - _reLat / MAX(_reDist, 1.0));
// //      //   yreDynGy := yreDynGy + _reRightY * _reRepulse * _creRightBias * _reDiffY / _reDist;
// //                //   * MAX(0.0, 1.0 - _reLat / MAX(_reDist, 1.0));
// // 			//   yreDynGy := yreDynGy +_reRightY + _reRepulse * _reDiffY / _reDist;
// //     //	END_IF
// // //END_IF
END_FOR

yreAusgangsTest := _reRepulse;

IF yboStop THEN yreSpeedFactor := 0.0; END_IF

END_FUNCTION_BLOCK

// ---- POUs/HAWinoCore/05_Bahnplanung/FB_RobotStateMachine.TcPOU
FUNCTION_BLOCK FB_RobotStateMachine
VAR_INPUT
    // ---------- MQTT inputs ----------
    xstMqttIn               : sMqttIn;                      // Full MQTT input struct (job + commands)
 
    // ---------- Robot status ----------
    xeRobotStatus           : RobotStatus;                  // Current robot status from controller
 
    // ---------- Map / algorithm feedback ----------
    xboMapsLoaded           : BOOL;                         // Maps successfully loaded → leave LoadMaps
    xboVectorTargetReached  : BOOL;                         // Vector algorithm has reached target
 
    // ---------- Coordinate array ----------
    xarstCoordinates        : ARRAY[0..29] OF sKoordinate;  // All station + RFID coordinates for this robot
 
    // ---------- Index inputs (set externally via GVL constants) ----------
    xinSourceIndex          : INT;                          // Array index of source station  (0..21)
	xinSourceDirectionIndex : INT;
    xinTargetIndex          : INT;                          // Array index of target station  (0..21)
	xinTargetDirectionIndex : INT;
    xinRfidSourceIndex      : INT;                          // Array index of RFID point at source (22..29)
    xinRfidTargetIndex      : INT;                          // Array index of RFID point at target (22..29)
    xinParkingIndex         : INT;                          // Array index of parking position (16..19)
    xinChargingIndex        : INT;                          // Array index of charging station (20..21)
 
    // ---------- Map ID inputs ----------
    xinMapSource            : INT;                          // Map ID for source station
    xinMapTarget            : INT;                          // Map ID for target station
    xinMapParking           : INT;                          // Map ID for parking position
	
	xreDistToGoal 			:REAL;
	xreDistFromGoal			:REAL;
	xboWSSensor				:BOOL;							//light switch for Thing
	xboAwayFromObstacle 	:BOOL;
	xinStatusOfChargin		: INT;
END_VAR
 
VAR_OUTPUT
    // ---------- Robot control ----------
    yeControl               : RobotControl;                 // Command to vector/position controller
 
    // ---------- Target position ----------
    ystTargetPosition       : sPosition;                    // Current target coordinates for controller
 
    // ---------- Map selection ----------
    yinTargetMap            : INT;                          // Active map ID for vector algorithm
 
    // ---------- MQTT outputs ----------
    ystMqttOut              : sMqttOut;                     // Full MQTT output struct
 
    // ---------- Diagnostics ----------
    yeCurrentState          : E_RobotState;                 // Current state (HMI / diagnostics)
	
	yeMqttTokenTargetId			:INT; 							//Current Token Request Target
	yboPassiveWait : BOOL;
	yboDriveAway : BOOL;
	yboCharging : BOOL;
	yinCharginStationID	: INT;
END_VAR
 
VAR
    // Active state
    eState                  : E_RobotState;
 
    // Previous-cycle values for rising-edge detection
    eStatusOld              : RobotStatus;
    boVectorOld             : BOOL;
    boRfidCompleteOld       : BOOL;
    boTokenGrantOld         : BOOL;
 
    // Rising-edge flags (TRUE for exactly one cycle)
    boPositionReached       : BOOL;     // RobotStatus transition → zielErreicht
    boVectorReached         : BOOL;     // xboVectorTargetReached rising edge
    boRfidComplete          : BOOL;     // boRFIDComplete rising edge
    boTokenGrant            : BOOL;     // boTokenGrant rising edge
	boJobIDOld				: INT;
	boNewJob				: BOOL;		//Job ID changed
	boCancelCharging		: BOOL;
	
	TONTokenRequestTime		: TON;
	TONGripperTime			: TON;
	TONChargingDelay		: TON;
	boErrorStandStill		: BOOL;
	eStateOld				: E_RobotState;
	eHelperStateOld			: E_RobotState;
	
	TONGripperEnable :TON;
END_VAR

VAR CONSTANT
	creDistanzForToken : REAL := 70;
	creDistanzForTokenRelease : REAL := 40;
	crePreTargetDistance : REAL := 100;
	ctiGripperTime 		: TIME := T#2.0S;
END_VAR

// ---------------------------------------------------------------------------
// Rising-edge detection
// ---------------------------------------------------------------------------
{region 'Edge'}
boPositionReached := (xeRobotStatus = RobotStatus.zielErreicht)
                     AND NOT (eStatusOld = RobotStatus.zielErreicht);
 
boVectorReached   := xboVectorTargetReached AND NOT boVectorOld;
 
boRfidComplete    := xstMqttIn.sCmd.boRFIDComplete AND NOT boRfidCompleteOld;
 
boTokenGrant      := xstMqttIn.sCmd.boTokenGrant   AND NOT boTokenGrantOld;
(*IF NOT( boJobIDOld = xstMqttIn.sJOB.inJobID) THEN
		boNewJob := TRUE;
	ELSE
		boNewJob := FALSE;
END_IF*)
	IF xstMqttIn.boNewJob AND ((eState = E_RobotState.Standby) OR (eState = E_RobotState.SelectMapParkPosition)) THEN
		boNewJob := TRUE;
	END_IF
	
	
IF xstMqttIn.sCmd.boCancelCharging THEN
	boCancelCharging := TRUE;
END_IF
{endregion}
{region 'Init'}
// Store previous values
eStatusOld        := xeRobotStatus;
boVectorOld       := xboVectorTargetReached;
boRfidCompleteOld := xstMqttIn.sCmd.boRFIDComplete;
boTokenGrantOld   := xstMqttIn.sCmd.boTokenGrant;
boJobIDOld 		  := xstMqttIn.sJOB.inJobID;
	
IF eState <> eHelperStateOld THEN
    eStateOld     := eHelperStateOld;
    eHelperStateOld := eState;
END_IF
 
// ---------------------------------------------------------------------------
// Reset cyclic outputs each scan (only re-set inside states that need them)
// ---------------------------------------------------------------------------
yeControl                                := RobotControl.idle;
ystMqttOut.sJobState.boWaitForRfidOut    := FALSE;
ystMqttOut.sJobState.boWaitForRfidIn     := FALSE;
ystMqttOut.sToken.boTokenRequest         := FALSE;
ystMqttOut.sToken.boTokenRelease         := FALSE;
ystMqttOut.sJobState.boJobAccepted       := FALSE;
ystMqttOut.sJobState.boWorkpiecePlaced   := FALSE;
 {endregion}
// ---------------------------------------------------------------------------
// STATE MACHINE – matches DrawIO diagram V2.1 exactly
// ---------------------------------------------------------------------------

// Stop
IF xeRobotStatus = RobotStatus.fehler OR xstMqttIn.sCmd.boStop THEN
	boErrorStandStill := TRUE;
	yeControl := RobotControl.idle;
END_IF
IF xeRobotStatus = RobotStatus.fehler THEN
	ystMqttOut.sError.boErrorControl := TRUE;
END_IF
IF xstMqttIn.sCmd.boReset OR xstMqttIn.sCmd.boJobReset AND (NOT ((eState = E_RobotState.WaitForChargingDone) OR (eState = E_RobotState.AtChargingStation))) THEN
	IF xstMqttIn.sCmd.boJobReset THEN //Hard Error
		eState := E_RobotState.SelectMapParkPosition;
	END_IF
	xstMqttIn.sJOB.inJobID := 0;
	boErrorStandStill := FALSE;
	yeControl :=  RobotControl.reset;
	ystMqttOut.sError.boErrorControl := FALSE;
	boNewJob := FALSE;
	RETURN;
ELSIF  xstMqttIn.sCmd.boJobReset AND ((eState = E_RobotState.AtChargingStation) OR (eState = E_RobotState.WaitForChargingDone)) THEN
	boCancelCharging := TRUE;
	xstMqttIn.sJOB.inJobID := 0;
	ystMqttOut.sError.boErrorControl := FALSE;
	boErrorStandStill := FALSE;
	boNewJob := FALSE;
END_IF



//Hard Error
(*IF xstMqttIn.sCmd.boJobReset THEN
	eState := E_RobotState.SelectMapParkPosition;
END_IF
*)

IF NOT boErrorStandStill THEN
{region 'StateMachine'}
CASE eState OF
{region 'Start'}
    // ------------------------------------------------------------------
    // LOAD MAPS
    // Initial state. Moves to Standby as soon as maps are loaded.
    // ------------------------------------------------------------------
    E_RobotState.LoadMaps:
        yeControl := RobotControl.idle;
        IF xboMapsLoaded THEN
            eState := E_RobotState.Standby;
        END_IF
 
    // ------------------------------------------------------------------
    // STANDBY
    // Ready and waiting for a new job (boStartJob via MQTT).
    // ------------------------------------------------------------------
    E_RobotState.Standby:
        yeControl := RobotControl.idle;
        ystMqttOut.sGeneralState.boReady := TRUE;
		Gripper.closeGripperCommand := FALSE;

        IF boNewJob THEN  //xstMqttIn.sCmd.boStartJob
			boNewJob := FALSE;
            eState := E_RobotState.CheckConfirmJob;
        END_IF
 
    // ------------------------------------------------------------------
    // CHECK / CONFIRM JOB
    // Signal job acceptance, then immediately select source map.
    // ------------------------------------------------------------------
    E_RobotState.CheckConfirmJob:
        ystMqttOut.sJobState.boJobAccepted := TRUE;
		 IF xstMqttIn.sCmd.boStartJob THEN  
            ystMqttOut.sGeneralState.boReady := FALSE;
			ystMqttOut.sJobState.boJobAccepted := FALSE;
			yinTargetMap := xinMapSource;
            eState := E_RobotState.SelectMapStart;
        END_IF
{endregion}
 {region 'Source'}
    // ------------------------------------------------------------------
    // SELECT MAP – SOURCE SIDE
    // Start vector algorithm towards source halt point.
    // Branch: halt point reached + job = parking → SelectMapParkPosition
    //         halt point reached + job ≠ parking → WaitPassiveSource
    //         vector not yet done               → WaitpointReachedSource
    // ------------------------------------------------------------------
    E_RobotState.SelectMapStart:
        yeControl    := RobotControl.vector;
 
 		IF ((xstMqttIn.sJOB.inDestination1 = 101) OR (xstMqttIn.sJOB.inDestination1 = 102) OR (xstMqttIn.sJOB.inDestination1 = 103) OR (xstMqttIn.sJOB.inDestination1 = 104)) THEN
			eState := E_RobotState.SelectMapParkPosition;
			 yinTargetMap               := xinMapParking;
		END_IF;
		IF (xstMqttIn.sJOB.inDestination1 = 201) OR (xstMqttIn.sJOB.inDestination1 = 202) THEN 
			eState := E_RobotState.AlgorithmPreviousSource;
			 yinTargetMap               := xinMapSource;
		END_IF
        
        IF xreDistToGoal < creDistanzForToken THEN
			eState := E_RobotState.WaitPassiveSource;
		END_IF
			
	(*		
            eState := E_RobotState.WaitPassiveSource;
        ELSE
            eState := E_RobotState.WaitpointReachedSource;
        END_IF
 *)
    // ------------------------------------------------------------------
    // WAITPOINT REACHED – SOURCE SIDE
    // Wait for Token
	//TODO: IMPlement Passive Wait here.
    // ------------------------------------------------------------------
    E_RobotState.WaitpointReachedSource:
        yeControl := RobotControl.vector;
		yboPassiveWait := TRUE;
        IF boTokenGrant THEN
			yboPassiveWait := FALSE;
            eState := E_RobotState.AlgorithmPreviousSource;
        END_IF
 
    // ------------------------------------------------------------------
    // WAIT PASSIVE – SOURCE SIDE
    // Halt point occupied. Request token and stop until granted.
		
	
    // ------------------------------------------------------------------
    E_RobotState.WaitPassiveSource:
        yeControl := RobotControl.vector;
        ystMqttOut.sToken.boTokenRequest := TRUE;
		yeMqttTokenTargetId := xinMapSource;
		
        IF boTokenGrant THEN
            eState := E_RobotState.AlgorithmPreviousSource;
		ELSIF TONTokenRequestTime.Q THEN
			eState := E_RobotState.WaitpointReachedSource;
        END_IF
 	
    // ------------------------------------------------------------------
    // ALGORITHM TO PREVIOUS TARGET – SOURCE SIDE
    // Resume movement after token received.
    // ------------------------------------------------------------------
    E_RobotState.AlgorithmPreviousSource:
        yeControl    := RobotControl.vector;
        yinTargetMap := xinMapSource;
        IF boVectorReached THEN
            eState := E_RobotState.DrivePoint2Align;//SwitchCoordinatesSource;
        END_IF
 
    // ------------------------------------------------------------------
    // SWITCH COORDINATES – SOURCE SIDE
    // Load source station coordinate from array, switch to position mode.
    // ------------------------------------------------------------------
//     E_RobotState.SwitchCoordinatesSource:
//         yeControl                      := RobotControl.position;
// 		
// 		IF ((xstMqttIn.sJOB.inDestination1 = 201) OR (xstMqttIn.sJOB.inDestination1 = 202)) THEN
// 			ystTargetPosition.reX          := REAL_TO_LREAL(xarstCoordinates[xinSourceIndex].rePosX);
//         	ystTargetPosition.reY          := REAL_TO_LREAL(xarstCoordinates[xinSourceIndex].rePosY)  - crePreTargetDistance;
// 		ELSE
//         	ystTargetPosition.reX          := REAL_TO_LREAL(xarstCoordinates[xinSourceIndex].rePosX) + (crePreTargetDistance * xinSourceDirectionIndex);
//         	ystTargetPosition.reY          := REAL_TO_LREAL(xarstCoordinates[xinSourceIndex].rePosY);
// 		END_IF
// 		
//         ystTargetPosition.reWinkel     := REAL_TO_LREAL(xarstCoordinates[xinSourceIndex].reWinkel);
//         IF boPositionReached THEN
//             eState := E_RobotState.DrivePoint1Align;
//         END_IF
 
    // ------------------------------------------------------------------
    // DRIVE TO POINT 1 + ALIGN  (approach point in front of source)
    // ------------------------------------------------------------------
    E_RobotState.DrivePoint1Align:
        yeControl := RobotControl.position;
        IF TRUE THEN //boPositionReached THEN
            eState := E_RobotState.DrivePoint2Align;
        END_IF
 
    // ------------------------------------------------------------------
    // DRIVE TO POINT 2 + ALIGN
    // Branch: job = charging (ID 3) → AtChargingStation
    //         normal                → AtStation
    // ------------------------------------------------------------------
    E_RobotState.DrivePoint2Align:
        yeControl := RobotControl.position;
		IF ((xstMqttIn.sJOB.inDestination1 = 201) OR (xstMqttIn.sJOB.inDestination1 = 202)) THEN
			//TODO Umschaltung Regler
			ystTargetPosition.reX          := REAL_TO_LREAL(xarstCoordinates[xinSourceIndex].rePosX);
        	ystTargetPosition.reY          := REAL_TO_LREAL(xarstCoordinates[xinSourceIndex].rePosY);
		ELSE
        	ystTargetPosition.reX          := REAL_TO_LREAL(xarstCoordinates[xinSourceIndex].rePosX);
        	ystTargetPosition.reY          := REAL_TO_LREAL(xarstCoordinates[xinSourceIndex].rePosY);
		END_IF
		ystTargetPosition.reWinkel     := REAL_TO_LREAL(xarstCoordinates[xinSourceIndex].reWinkel);
        IF ( xstMqttIn.boCharging1Connected AND (xstMqttIn.sJOB.inDestination1 = 201)) OR ( xstMqttIn.boCharging2Connected AND(xstMqttIn.sJOB.inDestination1 = 202)) THEN
				//charging – adapt as needed
                eState := E_RobotState.AtChargingStation;
         ELSIF boPositionReached THEN
                eState := E_RobotState.AtStation;
         END_IF
 
    // ------------------------------------------------------------------
    // AT CHARGING STATION
    // Position reached – now wait for charging to complete.
    // ------------------------------------------------------------------
    E_RobotState.AtChargingStation:
        yeControl := RobotControl.idle;
		yboCharging := TRUE;
		IF (xstMqttIn.sJOB.inDestination1 = 201) THEN
			yinCharginStationID := 1;
		ELSIF (xstMqttIn.sJOB.inDestination1 = 202) THEN
			yinCharginStationID := 2;	
		END_IF
		
        IF TRUE THEN//(xinStatusOfChargin = 1) THEN //TODO Connect with Charging Active
            eState := E_RobotState.WaitForChargingDone;
        END_IF
 
    // ------------------------------------------------------------------
    // WAIT FOR CHARGING DONE
    // Hold until boCancelCharging is received from MQTT.
    // ------------------------------------------------------------------
    E_RobotState.WaitForChargingDone:
		yboCharging := FALSE;
        yeControl := RobotControl.idle;
        ystMqttOut.sGeneralState.boCharging := TRUE;
        IF TONChargingDelay.Q THEN//AND (xinStatusOfChargin = 1) THEN //TODO Wait for canceled Charging
			boCancelCharging := FALSE;
            ystMqttOut.sGeneralState.boCharging := FALSE;
            eState := E_RobotState.DrivePoint1AfterCharge;
        END_IF
 
    // ------------------------------------------------------------------
    // DRIVE TO POINT 1 BEFORE STATION (after charging)
    // Returns to main flow via SelectMapParkPosition.
    // ------------------------------------------------------------------
    E_RobotState.DrivePoint1AfterCharge:
	     
        yeControl := RobotControl.vector;
		yboDriveAway := TRUE;
		(*ystTargetPosition.reX          := REAL_TO_LREAL(xarstCoordinates[xinSourceIndex].rePosX);
        ystTargetPosition.reY          := REAL_TO_LREAL(xarstCoordinates[xinSourceIndex].rePosY)  - crePreTargetDistance;
        ystTargetPosition.reWinkel     := REAL_TO_LREAL(xarstCoordinates[xinSourceIndex].reWinkel);*)
		
        IF xboAwayFromObstacle THEN
			yboDriveAway := FALSE;
            eState := E_RobotState.SelectMapParkPosition;
			 yinTargetMap               := xinMapParking;
        END_IF
 
    // ------------------------------------------------------------------
    // AT STATION
    // Branch: workpiece present → CloseGripper
    //         no workpiece      → DrivePoint1NoWorkpiece + error flag
    // ------------------------------------------------------------------
    E_RobotState.AtStation:
        yeControl := RobotControl.idle;
		
        IF xboWSSensor THEN
                eState := E_RobotState.CloseGripper;
		ELSE
                ystMqttOut.sError.boErrorNoWorkpiece := TRUE;
                eState := E_RobotState.DrivePoint1NoWorkpiece;
        END_IF
 
    // ------------------------------------------------------------------
    // CLOSE GRIPPER
    // Wait for workpiece-loaded confirmation before continuing.
    // ------------------------------------------------------------------
    E_RobotState.CloseGripper:
        yeControl := RobotControl.idle;
		Gripper.closeGripperCommand := TRUE;

		IF Gripper.state_out = CoreGripperControlState.Closed THEN
			ystMqttOut.sJobState.boTransportWorkpiece := TRUE;
            eState := E_RobotState.DrivePoint1WithWorkpiece;
// 		ELSIF TONGripperTime.Q THEN			// Backup, falls der Gripper nicht schließt									<-------------------------------------------------------------------Hier einmal
//             eState := E_RobotState.Standby;	// Hier noch in einen Sinvolleren Zustand springen
		END_IF
    
    // ------------------------------------------------------------------
    // DRIVE TO POINT 1 – NO WORKPIECE
    // Workpiece missing path → directly to SelectMapParkPosition.
    // ------------------------------------------------------------------
    E_RobotState.DrivePoint1NoWorkpiece:
        yeControl := RobotControl.vector;
		yboDriveAway := TRUE;
        (*ystTargetPosition.reX          := REAL_TO_LREAL(xarstCoordinates[xinSourceIndex].rePosX) + (crePreTargetDistance * xinSourceDirectionIndex);
        ystTargetPosition.reY          := REAL_TO_LREAL(xarstCoordinates[xinSourceIndex].rePosY);
        ystTargetPosition.reWinkel     := REAL_TO_LREAL(xarstCoordinates[xinSourceIndex].reWinkel);*)
        IF xboAwayFromObstacle THEN
			yboDriveAway := FALSE;
			ystMqttOut.sError.boErrorNoWorkpiece := FALSE;
            eState := E_RobotState.SelectMapParkPosition;
			 yinTargetMap               := xinMapParking;
        END_IF
 
    // ------------------------------------------------------------------
    // DRIVE TO POINT 1 – WITH WORKPIECE
    // Normal return path WITH workpiece → continue to point 3.
    // ------------------------------------------------------------------
    E_RobotState.DrivePoint1WithWorkpiece:
		yeControl    := RobotControl.vector; //test for driving back insted of point
		yboDriveAway := TRUE;
        //yeControl := RobotControl.position;
		(*ystTargetPosition.reX          := REAL_TO_LREAL(xarstCoordinates[xinSourceIndex].rePosX) + (crePreTargetDistance * xinSourceDirectionIndex);
        ystTargetPosition.reY          := REAL_TO_LREAL(xarstCoordinates[xinSourceIndex].rePosY);
        ystTargetPosition.reWinkel     := REAL_TO_LREAL(xarstCoordinates[xinSourceIndex].reWinkel);*)
        IF xboAwayFromObstacle THEN//boPositionReached THEN
			yboDriveAway := FALSE;
            eState := E_RobotState.DrivePoint4;//DrivePoint3Align;
        END_IF
 
    // ------------------------------------------------------------------
    // DRIVE TO POINT 3 + ALIGN
    // ------------------------------------------------------------------
//     E_RobotState.DrivePoint3Align:
//         yeControl := RobotControl.position;
// 		ystTargetPosition.reX      := REAL_TO_LREAL(xarstCoordinates[xinRfidSourceIndex].rePosX)+ (crePreTargetDistance * xinSourceDirectionIndex);
//         ystTargetPosition.reY      := REAL_TO_LREAL(xarstCoordinates[xinRfidSourceIndex].rePosY);
//         ystTargetPosition.reWinkel := REAL_TO_LREAL(xarstCoordinates[xinRfidSourceIndex].reWinkel);
//         IF boPositionReached THEN//boPositionReached THEN
//             eState := E_RobotState.DrivePoint4;
//         END_IF
//  
    // ------------------------------------------------------------------
    // DRIVE TO POINT 4
    // Load RFID source coordinate before transitioning to RFID scan.
    // ------------------------------------------------------------------
    E_RobotState.DrivePoint4:
        yeControl := RobotControl.position;
		ystTargetPosition.reX      := REAL_TO_LREAL(xarstCoordinates[xinRfidSourceIndex].rePosX);
        ystTargetPosition.reY      := REAL_TO_LREAL(xarstCoordinates[xinRfidSourceIndex].rePosY);
        ystTargetPosition.reWinkel := REAL_TO_LREAL(xarstCoordinates[xinRfidSourceIndex].reWinkel);
		IF boPositionReached THEN
            eState := E_RobotState.ScanRFIDSource;
        END_IF
 
    // ------------------------------------------------------------------
    // SCAN RFID – SOURCE
    // Signal "waiting for RFID out" to controller. Wait for boRFIDComplete.
    // ------------------------------------------------------------------
    E_RobotState.ScanRFIDSource:
        yeControl := RobotControl.idle;
		ystMqttOut.sJobState.boWaitForRfidOut := TRUE;
        
        IF boRFIDComplete THEN
			ystMqttOut.sJobState.boWaitForRfidOut := FALSE;
            eState := E_RobotState.DrivePoint3ToTarget;
        END_IF
 
    // ------------------------------------------------------------------
    // DRIVE TO POINT 3 TOWARDS TARGET
    // ------------------------------------------------------------------
    E_RobotState.DrivePoint3ToTarget:
        (*yeControl := RobotControl.position;
		ystTargetPosition.reX      := REAL_TO_LREAL(xarstCoordinates[xinRfidSourceIndex].rePosX)+ (crePreTargetDistance * xinSourceDirectionIndex);
        ystTargetPosition.reY      := REAL_TO_LREAL(xarstCoordinates[xinRfidSourceIndex].rePosY);
        ystTargetPosition.reWinkel := REAL_TO_LREAL(xarstCoordinates[xinRfidSourceIndex].reWinkel);*)
		yeControl := RobotControl.vector;
		yboDriveAway := TRUE;
        IF xboAwayFromObstacle THEN
			yboDriveAway := FALSE;
            eState := E_RobotState.SelectMapTarget;
			yinTargetMap := xinMapTarget;
        END_IF
 {endregion}
    // ------------------------------------------------------------------
    // SELECT MAP – TARGET SIDE
    // Start vector algorithm towards target halt point.
    // Normal path → WaitpointReachedTarget
    // Side path (distance below threshold & no token) → WaitPassiveTarget
    // ------------------------------------------------------------------
{region 'Target'}
    E_RobotState.SelectMapTarget:
        yinTargetMap := xinMapTarget;
        yeControl    := RobotControl.vector;
		
		IF ((xinMapSource = 2) AND (xinMapTarget = 3)) OR
		((xinMapSource = 4) AND (xinMapTarget = 5)) OR
		((xinMapSource = 6) AND (xinMapTarget = 7)) OR
		((xinMapSource = 3) AND (xinMapTarget = 2)) OR
		((xinMapSource = 5) AND (xinMapTarget = 4)) OR
		((xinMapSource = 7) AND (xinMapTarget = 6)) THEN
			ystMqttOut.sToken.boTokenRelease := TRUE;
		END_IF;
		
		IF xreDistFromGoal > creDistanzForTokenRelease THEN
			ystMqttOut.sToken.boTokenRelease := TRUE;
		END_IF
		 IF xreDistToGoal < creDistanzForToken THEN
			eState := E_RobotState.WaitpointReachedTarget;
		END_IF
		
	
 
    // ------------------------------------------------------------------
    // WAITPOINT REACHED – TARGET SIDE
    // ------------------------------------------------------------------
    E_RobotState.WaitpointReachedTarget:
        yeControl := RobotControl.vector;
		ystMqttOut.sToken.boTokenRequest := TRUE;
		yeMqttTokenTargetId := xinMapTarget;
        IF boTokenGrant THEN 
			ystMqttOut.sToken.boTokenRequest := FALSE;
            eState := E_RobotState.AlgorithmPreviousTarget;
		ELSIF TONTokenRequestTime.Q THEN
			eState := E_RobotState.WaitPassiveTarget;
        END_IF
 
    // ------------------------------------------------------------------
    // WAIT PASSIVE – TARGET SIDE
    // Halt point occupied. Request token, stop until granted.
    // ------------------------------------------------------------------
    E_RobotState.WaitPassiveTarget:
        yeControl := RobotControl.vector;
		yboPassiveWait := TRUE;
        IF boTokenGrant THEN
			yboPassiveWait := FALSE;
			ystMqttOut.sToken.boTokenRequest := FALSE;
            eState := E_RobotState.AlgorithmPreviousTarget;
        END_IF
 
